PROGRAM C03_AlarmMessageControl
VAR
	bAlarmGroup0Reset 		:BOOL;
	bAlarmGroup1Reset 		:BOOL;
	bAlarmGroup2Reset 		:BOOL;
	bAlarmGroup3Reset 		:BOOL;
	bAlarmGroup4Reset 		:BOOL;
	bAlarmGroup5Reset 		:BOOL;
	bAlarmGroup6Reset 		:BOOL;
	bAlarmGroup7Reset 		:BOOL;

	fbMsg_GroupPriority0	:FB_ALARM_GroupManagment;
	fbMsg_GroupPriority1	:FB_ALARM_GroupManagment;
	fbMsg_GroupPriority2	:FB_ALARM_GroupManagment;
	fbMsg_GroupPriority3	:FB_ALARM_GroupManagment;
	fbMsg_GroupPriority4	:FB_ALARM_GroupManagment;
	fbMsg_GroupPriority5	:FB_ALARM_GroupManagment;
	fbMsg_GroupPriority6	:FB_ALARM_GroupManagment;
	fbMsg_GroupPriority7	:FB_ALARM_GroupManagment;

	fbLogTable							: FB_ALARM_LogTable;
	//fbOutputDB						: FB_ALARM_OutputDB;

	aAlarmPulse						: ARRAY[0..255] OF TP;
	aTorqueStartDelayTimer			: ARRAY[1..cMAX_PROFINET_DRIVES] OF TON;

	nAlarmIndex						: INT;
	aMsgGroupStartIndex				: ARRAY[0..10] OF INT;

	bGeneralSystemAlarmActive		: BOOL;		(*Message type 0*)
	bEUCASubsytemAlarmActive		: BOOL;		(*Message type 1*)
	bTPDSubsytemAlarmActive			: BOOL;		(*Message type 2*)
	bExternalAlarmActive			: BOOL;		(*Message type 3*)

	bSpare04AlarmActive				: BOOL;		(*Message type 4*)
	bSpare05AlarmActive				: BOOL;		(*Message type 5*)
	bSpare06AlarmActive				: BOOL;		(*Message type 6*)
	bSpare07AlarmActive				: BOOL;		(*Message type 7*)

	bGeneralSystemWarningActive		: BOOL;		(*Message type 8*)
	bEUCASubsytemWarningActive		: BOOL;		(*Message type 9*)
	bTPDSubsytemWarningActive		: BOOL;		(*Message type 10*)
	bExternalWarningActive			: BOOL;		(*Message type 11*)

	bSpare12WarningActive			: BOOL;		(*Message type 12*)
	bSpare13WarningActive			: BOOL;		(*Message type 13*)
	bSpare14WarningActive			: BOOL;		(*Message type 14*)
	bSpare15WarningActive			: BOOL;		(*Message type 15*)

END_VAR
VAR // added by the converter: edge detectors and wires of the graphical bodies
    _w1, _w2, _w3, _w4, _w5, _w6, _w7, _w8 : BOOL;
END_VAR

(****************************************************************************************)
(*
bAlarmTrigger - set true to activate message
nCategoryNo - message category number (for future purpose)
nMessageTypeNo - message type number determine active message type flag
sTextMessage - message description shown in HMI
tAlarmTimout - message became active after time delay
bAlarmDefinitionEnable - enable message block executing
bInhibitReset - set acknowledge to reset/confirm active message 
*)
(****************************************************************************************)

MsgReset();
nAlarmIndex := 0;

(****************************************************************************************)

aMsgGroupStartIndex[0] := nAlarmIndex;
Msg_000_033_General();

aMsgGroupStartIndex[1] := nAlarmIndex;
Msg_034_074_Cameras();

aMsgGroupStartIndex[2] := nAlarmIndex;
Msg_075_126_Process();

aMsgGroupStartIndex[3] := nAlarmIndex;
Msg_127_150_Sensors();

aMsgGroupStartIndex[4] := nAlarmIndex;
Msg_151_179_Doors();

aMsgGroupStartIndex[5] := nAlarmIndex;
Msg_180_200_Motors();

aMsgGroupStartIndex[6] := nAlarmIndex;
Msg_201_208_Interface();

aMsgGroupStartIndex[7] := nAlarmIndex;
Msg_209_237_Labellers();

aMsgGroupStartIndex[8] := nAlarmIndex;
Msg_238_243_Spare();

aMsgGroupStartIndex[9] := nAlarmIndex;
Msg_244_253_DB();

aMsgGroupStartIndex[10] := nAlarmIndex;
Msg_254_255_Reserved();

(****************************************************************************************)

fbMsg_GroupPriority0	(

	stAlarms 				:= gMessage.aAlarms[0],
	stAlarmsSettings		:= gMessage.aAlarmsSettings[0]

					);
(****************************************************************************************)

fbMsg_GroupPriority1	(

	stAlarms 				:= gMessage.aAlarms[1],
	stAlarmsSettings		:= gMessage.aAlarmsSettings[1],

					);
(****************************************************************************************)

fbMsg_GroupPriority2	(

	stAlarms 				:= gMessage.aAlarms[2],
	stAlarmsSettings		:= gMessage.aAlarmsSettings[2]

					);
(****************************************************************************************)

fbMsg_GroupPriority3	(

	stAlarms 				:= gMessage.aAlarms[3],
	stAlarmsSettings		:= gMessage.aAlarmsSettings[3],

					);
(****************************************************************************************)

fbMsg_GroupPriority4		(

	stAlarms 				:= gMessage.aAlarms[4],
	stAlarmsSettings		:= gMessage.aAlarmsSettings[4]

					);
(****************************************************************************************)

fbMsg_GroupPriority5	(

	stAlarms 				:= gMessage.aAlarms[5],
	stAlarmsSettings		:= gMessage.aAlarmsSettings[5]

					);
(****************************************************************************************)

fbMsg_GroupPriority6	(

	stAlarms 				:= gMessage.aAlarms[6],
	stAlarmsSettings		:= gMessage.aAlarmsSettings[6]

					);
(****************************************************************************************)

fbMsg_GroupPriority7	(

	stAlarms 				:= gMessage.aAlarms[7],
	stAlarmsSettings		:= gMessage.aAlarmsSettings[7]

					);
(**************************************************************************************************)
(**************************** **********Alarms Logger***********************************************)
(**************************************************************************************************)

fbLogTable(
			bResetActive		:= gDevice.stMetsStatus.bShortReset,
			stAlarmTable		:= gMessage.stAlarmTable,
			aAlarms 			:= gMessage.aAlarms,
			aAlarmsSettings		:= gMessage.aAlarmsSettings,
			stCTDateTime		:= gDevice.stMetsStatus.stCTDateTime
		);
		
(*fbOutputDB(
	bSystemTimeValid		:= gDevice.stMetsStatus.bSystemTimeValid,
	stCTDateTime			:= gDevice.stMetsStatus.stCTDateTime,
	nAppOnlineChangeCnt 	:= gDevice.stPLCAppSys.OnlineChangeCnt,
	stAlarmTable			:= gMessage.stAlarmTable,
	stMachineConfig			:= gDevice.stMachineConfig
	);
*)
(**************************************************************************************************)
(**************************** **********Fault Monitor***********************************************)
(**************************************************************************************************)

IF 	gMessage.aAlarms[0].nMessageType.0	OR
	gMessage.aAlarms[1].nMessageType.0	OR
	gMessage.aAlarms[2].nMessageType.0	OR
	gMessage.aAlarms[3].nMessageType.0	OR
	gMessage.aAlarms[4].nMessageType.0	OR
	gMessage.aAlarms[5].nMessageType.0	OR
	gMessage.aAlarms[6].nMessageType.0	OR
	gMessage.aAlarms[7].nMessageType.0	THEN

		gMessage.stAlarmStatus.bGeneralSystemAlarmActive	:=	TRUE;
ELSE
		gMessage.stAlarmStatus.bGeneralSystemAlarmActive	:= 	FALSE;
END_IF

IF 	gMessage.aAlarms[0].nMessageType.1	OR
	gMessage.aAlarms[1].nMessageType.1	OR
	gMessage.aAlarms[2].nMessageType.1	OR
	gMessage.aAlarms[3].nMessageType.1	OR
	gMessage.aAlarms[4].nMessageType.1	OR
	gMessage.aAlarms[5].nMessageType.1	OR
	gMessage.aAlarms[6].nMessageType.1	OR
	gMessage.aAlarms[7].nMessageType.1	THEN

		gMessage.stAlarmStatus.bEUCASubsytemAlarmActive	:=	TRUE;
ELSE
		gMessage.stAlarmStatus.bEUCASubsytemAlarmActive	:= 	FALSE;
END_IF

IF 	gMessage.aAlarms[0].nMessageType.2	OR
	gMessage.aAlarms[1].nMessageType.2	OR
	gMessage.aAlarms[2].nMessageType.2	OR
	gMessage.aAlarms[3].nMessageType.2	OR
	gMessage.aAlarms[4].nMessageType.2	OR
	gMessage.aAlarms[5].nMessageType.2	OR
	gMessage.aAlarms[6].nMessageType.2	OR
	gMessage.aAlarms[7].nMessageType.2	THEN

		gMessage.stAlarmStatus.bTPDSubsytemAlarmActive	:=	TRUE;
ELSE
		gMessage.stAlarmStatus.bTPDSubsytemAlarmActive	:= 	FALSE;
END_IF

IF 	gMessage.aAlarms[0].nMessageType.3	OR
	gMessage.aAlarms[1].nMessageType.3	OR
	gMessage.aAlarms[2].nMessageType.3	OR
	gMessage.aAlarms[3].nMessageType.3	OR
	gMessage.aAlarms[4].nMessageType.3	OR
	gMessage.aAlarms[5].nMessageType.3	OR
	gMessage.aAlarms[6].nMessageType.3	OR
	gMessage.aAlarms[7].nMessageType.3	THEN

		gMessage.stAlarmStatus.bExternalAlarmActive	:=	TRUE;
ELSE
		gMessage.stAlarmStatus.bExternalAlarmActive	:= 	FALSE;
END_IF

IF 	gMessage.aAlarms[0].nMessageType.4	OR
	gMessage.aAlarms[1].nMessageType.4	OR
	gMessage.aAlarms[2].nMessageType.4	OR
	gMessage.aAlarms[3].nMessageType.4	OR
	gMessage.aAlarms[4].nMessageType.4	OR
	gMessage.aAlarms[5].nMessageType.4	OR
	gMessage.aAlarms[6].nMessageType.4	OR
	gMessage.aAlarms[7].nMessageType.4	THEN

		gMessage.stAlarmStatus.bSpare04AlarmActive	:=	TRUE;
ELSE
		gMessage.stAlarmStatus.bSpare04AlarmActive	:= 	FALSE;
END_IF

IF 	gMessage.aAlarms[0].nMessageType.5	OR
	gMessage.aAlarms[1].nMessageType.5	OR
	gMessage.aAlarms[2].nMessageType.5	OR
	gMessage.aAlarms[3].nMessageType.5	OR
	gMessage.aAlarms[4].nMessageType.5	OR
	gMessage.aAlarms[5].nMessageType.5	OR
	gMessage.aAlarms[6].nMessageType.5	OR
	gMessage.aAlarms[7].nMessageType.5	THEN

		gMessage.stAlarmStatus.bSpare05AlarmActive	:=	TRUE;
ELSE
		gMessage.stAlarmStatus.bSpare05AlarmActive	:= 	FALSE;
END_IF

IF 	gMessage.aAlarms[0].nMessageType.6	OR
	gMessage.aAlarms[1].nMessageType.6	OR
	gMessage.aAlarms[2].nMessageType.6	OR
	gMessage.aAlarms[3].nMessageType.6	OR
	gMessage.aAlarms[4].nMessageType.6	OR
	gMessage.aAlarms[5].nMessageType.6	OR
	gMessage.aAlarms[6].nMessageType.6	OR
	gMessage.aAlarms[7].nMessageType.6	THEN

		gMessage.stAlarmStatus.bSpare06AlarmActive	:=	TRUE;
ELSE
		gMessage.stAlarmStatus.bSpare06AlarmActive	:= 	FALSE;
END_IF

IF 	gMessage.aAlarms[0].nMessageType.7	OR
	gMessage.aAlarms[1].nMessageType.7	OR
	gMessage.aAlarms[2].nMessageType.7	OR
	gMessage.aAlarms[3].nMessageType.7	OR
	gMessage.aAlarms[4].nMessageType.7	OR
	gMessage.aAlarms[5].nMessageType.7	OR
	gMessage.aAlarms[6].nMessageType.7	OR
	gMessage.aAlarms[7].nMessageType.7	THEN

		gMessage.stAlarmStatus.bSpare07AlarmActive	:=	TRUE;
ELSE
		gMessage.stAlarmStatus.bSpare07AlarmActive	:= 	FALSE;
END_IF


IF 	gMessage.aAlarms[0].nMessageType.8	OR
	gMessage.aAlarms[1].nMessageType.8	OR
	gMessage.aAlarms[2].nMessageType.8	OR
	gMessage.aAlarms[3].nMessageType.8	OR
	gMessage.aAlarms[4].nMessageType.8	OR
	gMessage.aAlarms[5].nMessageType.8	OR
	gMessage.aAlarms[6].nMessageType.8	OR
	gMessage.aAlarms[7].nMessageType.8	THEN

		gMessage.stAlarmStatus.bGeneralSystemWarningActive	:=	TRUE;
ELSE
		gMessage.stAlarmStatus.bGeneralSystemWarningActive	:= 	FALSE;
END_IF

IF 	gMessage.aAlarms[0].nMessageType.9	OR
	gMessage.aAlarms[1].nMessageType.9	OR
	gMessage.aAlarms[2].nMessageType.9	OR
	gMessage.aAlarms[3].nMessageType.9	OR
	gMessage.aAlarms[4].nMessageType.9	OR
	gMessage.aAlarms[5].nMessageType.9	OR
	gMessage.aAlarms[6].nMessageType.9	OR
	gMessage.aAlarms[7].nMessageType.9	THEN

		gMessage.stAlarmStatus.bEUCASubsytemWarningActive	:=	TRUE;
ELSE
		gMessage.stAlarmStatus.bEUCASubsytemWarningActive	:= 	FALSE;
END_IF

IF 	gMessage.aAlarms[0].nMessageType.10	OR
	gMessage.aAlarms[1].nMessageType.10	OR
	gMessage.aAlarms[2].nMessageType.10	OR
	gMessage.aAlarms[3].nMessageType.10	OR
	gMessage.aAlarms[4].nMessageType.10	OR
	gMessage.aAlarms[5].nMessageType.10	OR
	gMessage.aAlarms[6].nMessageType.10	OR
	gMessage.aAlarms[7].nMessageType.10	THEN

		gMessage.stAlarmStatus.bTPDSubsytemWarningActive	:=	TRUE;
ELSE
		gMessage.stAlarmStatus.bTPDSubsytemWarningActive	:= 	FALSE;
END_IF

IF 	gMessage.aAlarms[0].nMessageType.11	OR
	gMessage.aAlarms[1].nMessageType.11	OR
	gMessage.aAlarms[2].nMessageType.11	OR
	gMessage.aAlarms[3].nMessageType.11	OR
	gMessage.aAlarms[4].nMessageType.11	OR
	gMessage.aAlarms[5].nMessageType.11	OR
	gMessage.aAlarms[6].nMessageType.11	OR
	gMessage.aAlarms[7].nMessageType.11	THEN

		gMessage.stAlarmStatus.bExternalWarningActive	:=	TRUE;
ELSE
		gMessage.stAlarmStatus.bExternalWarningActive	:= 	FALSE;
END_IF

IF 	gMessage.aAlarms[0].nMessageType.12	OR
	gMessage.aAlarms[1].nMessageType.12	OR
	gMessage.aAlarms[2].nMessageType.12	OR
	gMessage.aAlarms[3].nMessageType.12	OR
	gMessage.aAlarms[4].nMessageType.12	OR
	gMessage.aAlarms[5].nMessageType.12	OR
	gMessage.aAlarms[6].nMessageType.12	OR
	gMessage.aAlarms[7].nMessageType.12	THEN

		gMessage.stAlarmStatus.bSpare12WarningActive	:=	TRUE;
ELSE
		gMessage.stAlarmStatus.bSpare12WarningActive	:= 	FALSE;
END_IF

IF 	gMessage.aAlarms[0].nMessageType.13	OR
	gMessage.aAlarms[1].nMessageType.13	OR
	gMessage.aAlarms[2].nMessageType.13	OR
	gMessage.aAlarms[3].nMessageType.13	OR
	gMessage.aAlarms[4].nMessageType.13	OR
	gMessage.aAlarms[5].nMessageType.13	OR
	gMessage.aAlarms[6].nMessageType.13	OR
	gMessage.aAlarms[7].nMessageType.13	THEN

		gMessage.stAlarmStatus.bSpare13WarningActive	:=	TRUE;
ELSE
		gMessage.stAlarmStatus.bSpare13WarningActive	:= 	FALSE;
END_IF

IF 	gMessage.aAlarms[0].nMessageType.14	OR
	gMessage.aAlarms[1].nMessageType.14	OR
	gMessage.aAlarms[2].nMessageType.14	OR
	gMessage.aAlarms[3].nMessageType.14	OR
	gMessage.aAlarms[4].nMessageType.14	OR
	gMessage.aAlarms[5].nMessageType.14	OR
	gMessage.aAlarms[6].nMessageType.14	OR
	gMessage.aAlarms[7].nMessageType.14	THEN

		gMessage.stAlarmStatus.bSpare14WarningActive	:=	TRUE;
ELSE
		gMessage.stAlarmStatus.bSpare14WarningActive	:= 	FALSE;
END_IF

IF 	gMessage.aAlarms[0].nMessageType.15	OR
	gMessage.aAlarms[1].nMessageType.15	OR
	gMessage.aAlarms[2].nMessageType.15	OR
	gMessage.aAlarms[3].nMessageType.15	OR
	gMessage.aAlarms[4].nMessageType.15	OR
	gMessage.aAlarms[5].nMessageType.15	OR
	gMessage.aAlarms[6].nMessageType.15	OR
	gMessage.aAlarms[7].nMessageType.15	THEN

		gMessage.stAlarmStatus.bSpare15WarningActive	:=	TRUE;
ELSE
		gMessage.stAlarmStatus.bSpare15WarningActive	:= 	FALSE;
END_IF

(**************************************************************************************************)
(**********************************Group Fault Monitor**********************************************)
(**************************************************************************************************)

(*Message type from 0 to 3 are set up as alarms - if modyfie it is neccesary change alarm definition F_ALARM_SetDefinition for AutoReset flag*)

IF 	gMessage.stAlarmStatus.bGeneralSystemAlarmActive 		OR
	gMessage.stAlarmStatus.bEUCASubsytemAlarmActive 		OR
	gMessage.stAlarmStatus.bTPDSubsytemAlarmActive			OR
	gMessage.stAlarmStatus.bExternalAlarmActive				OR
	gMessage.stAlarmStatus.bSpare04AlarmActive 				OR
	gMessage.stAlarmStatus.bSpare05AlarmActive 				OR
	gMessage.stAlarmStatus.bSpare06AlarmActive				OR
	gMessage.stAlarmStatus.bSpare07AlarmActive				THEN

		gMessage.stAlarmStatus.bNoActiveAlarms	:=	FALSE;
ELSE
		gMessage.stAlarmStatus.bNoActiveAlarms	:=	TRUE;
END_IF

(*Message type from 4 to 7 are set up as warnings - if modyfie it is neccesary change alarm definition F_ALARM_SetDefinition for AutoReset flag*)

IF 	gMessage.stAlarmStatus.bGeneralSystemWarningActive 		OR
	gMessage.stAlarmStatus.bEUCASubsytemWarningActive 	OR
	gMessage.stAlarmStatus.bTPDSubsytemWarningActive		OR
	gMessage.stAlarmStatus.bExternalWarningActive			OR
	gMessage.stAlarmStatus.bSpare12WarningActive 			OR
	gMessage.stAlarmStatus.bSpare13WarningActive 			OR
	gMessage.stAlarmStatus.bSpare14WarningActive			OR
	gMessage.stAlarmStatus.bSpare15WarningActive			THEN

		gMessage.stAlarmStatus.bNoActiveWarrnings	:=	FALSE;
ELSE
		gMessage.stAlarmStatus.bNoActiveWarrnings	:=	TRUE;
END_IF

ACTION Msg_000_033_General:
// note: this text did not pass the execution check against the stored diagram
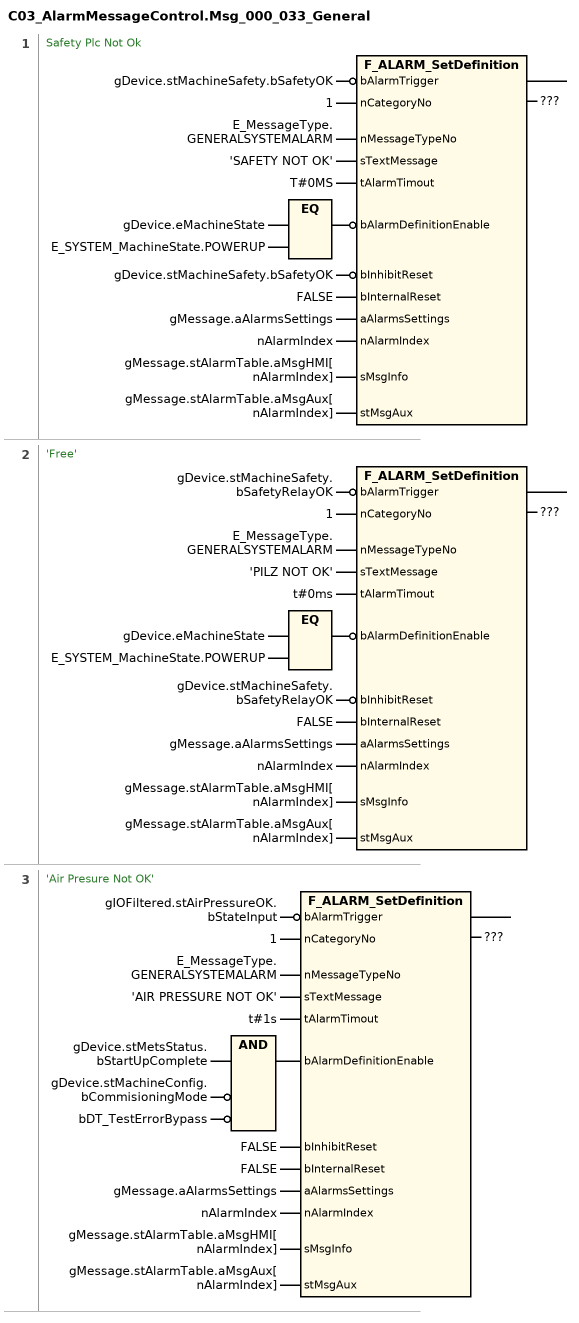
// NETWORK 1
//  Safety Plc Not Ok
F_ALARM_SetDefinition(bAlarmTrigger := NOT gDevice.stMachineSafety.bSafetyOK, nCategoryNo := 1, nMessageTypeNo := E_MessageType.GENERALSYSTEMALARM, sTextMessage := 'SAFETY NOT OK', tAlarmTimout := T#0MS, bAlarmDefinitionEnable := NOT (gDevice.eMachineState = E_SYSTEM_MachineState.POWERUP), bInhibitReset := NOT gDevice.stMachineSafety.bSafetyOK, bInternalReset := FALSE, aAlarmsSettings := gMessage.aAlarmsSettings, nAlarmIndex := nAlarmIndex, sMsgInfo := gMessage.stAlarmTable.aMsgHMI[nAlarmIndex], stMsgAux := gMessage.stAlarmTable.aMsgAux[nAlarmIndex]);

// NETWORK 2
// 'Free'
F_ALARM_SetDefinition(bAlarmTrigger := NOT gDevice.stMachineSafety.bSafetyRelayOK, nCategoryNo := 1, nMessageTypeNo := E_MessageType.GENERALSYSTEMALARM, sTextMessage := 'PILZ NOT OK', tAlarmTimout := t#0ms, bAlarmDefinitionEnable := NOT (gDevice.eMachineState = E_SYSTEM_MachineState.POWERUP), bInhibitReset := NOT gDevice.stMachineSafety.bSafetyRelayOK, bInternalReset := FALSE, aAlarmsSettings := gMessage.aAlarmsSettings, nAlarmIndex := nAlarmIndex, sMsgInfo := gMessage.stAlarmTable.aMsgHMI[nAlarmIndex], stMsgAux := gMessage.stAlarmTable.aMsgAux[nAlarmIndex]);

// NETWORK 3
// 'Air Presure Not OK'
F_ALARM_SetDefinition(bAlarmTrigger := NOT gIOFiltered.stAirPressureOK.bStateInput, nCategoryNo := 1, nMessageTypeNo := E_MessageType.GENERALSYSTEMALARM, sTextMessage := 'AIR PRESSURE NOT OK', tAlarmTimout := t#1s, bAlarmDefinitionEnable := gDevice.stMetsStatus.bStartUpComplete AND NOT gDevice.stMachineConfig.bCommisioningMode AND NOT bDT_TestErrorBypass, bInhibitReset := FALSE, bInternalReset := FALSE, aAlarmsSettings := gMessage.aAlarmsSettings, nAlarmIndex := nAlarmIndex, sMsgInfo := gMessage.stAlarmTable.aMsgHMI[nAlarmIndex], stMsgAux := gMessage.stAlarmTable.aMsgAux[nAlarmIndex]);

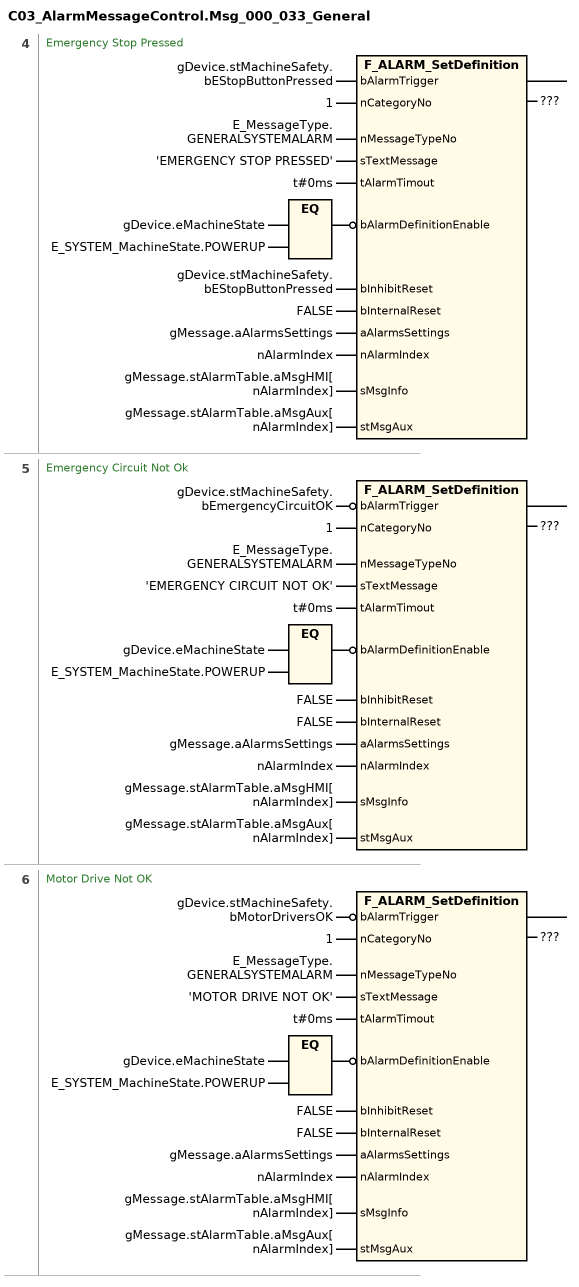
// NETWORK 4
// 					Emergency Stop Pressed
//
//
F_ALARM_SetDefinition(bAlarmTrigger := gDevice.stMachineSafety.bEStopButtonPressed, nCategoryNo := 1, nMessageTypeNo := E_MessageType.GENERALSYSTEMALARM, sTextMessage := 'EMERGENCY STOP PRESSED', tAlarmTimout := t#0ms, bAlarmDefinitionEnable := NOT (gDevice.eMachineState = E_SYSTEM_MachineState.POWERUP), bInhibitReset := gDevice.stMachineSafety.bEStopButtonPressed, bInternalReset := FALSE, aAlarmsSettings := gMessage.aAlarmsSettings, nAlarmIndex := nAlarmIndex, sMsgInfo := gMessage.stAlarmTable.aMsgHMI[nAlarmIndex], stMsgAux := gMessage.stAlarmTable.aMsgAux[nAlarmIndex]);

// NETWORK 5
// 					Emergency Circuit Not Ok
//
//
F_ALARM_SetDefinition(bAlarmTrigger := NOT gDevice.stMachineSafety.bEmergencyCircuitOK, nCategoryNo := 1, nMessageTypeNo := E_MessageType.GENERALSYSTEMALARM, sTextMessage := 'EMERGENCY CIRCUIT NOT OK', tAlarmTimout := t#0ms, bAlarmDefinitionEnable := NOT (gDevice.eMachineState = E_SYSTEM_MachineState.POWERUP), bInhibitReset := FALSE, bInternalReset := FALSE, aAlarmsSettings := gMessage.aAlarmsSettings, nAlarmIndex := nAlarmIndex, sMsgInfo := gMessage.stAlarmTable.aMsgHMI[nAlarmIndex], stMsgAux := gMessage.stAlarmTable.aMsgAux[nAlarmIndex]);

// NETWORK 6
// 					Motor Drive Not OK
//
//
F_ALARM_SetDefinition(bAlarmTrigger := NOT gDevice.stMachineSafety.bMotorDriversOK, nCategoryNo := 1, nMessageTypeNo := E_MessageType.GENERALSYSTEMALARM, sTextMessage := 'MOTOR DRIVE NOT OK', tAlarmTimout := t#0ms, bAlarmDefinitionEnable := NOT (gDevice.eMachineState = E_SYSTEM_MachineState.POWERUP), bInhibitReset := FALSE, bInternalReset := FALSE, aAlarmsSettings := gMessage.aAlarmsSettings, nAlarmIndex := nAlarmIndex, sMsgInfo := gMessage.stAlarmTable.aMsgHMI[nAlarmIndex], stMsgAux := gMessage.stAlarmTable.aMsgAux[nAlarmIndex]);

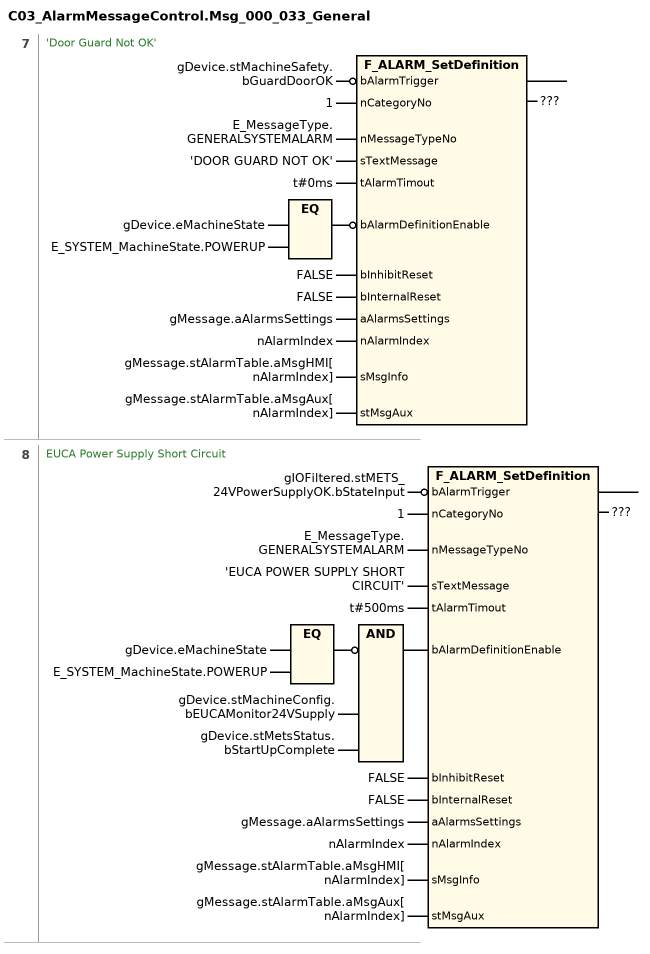
// NETWORK 7
// 					'Door Guard Not OK'
//
//
F_ALARM_SetDefinition(bAlarmTrigger := NOT gDevice.stMachineSafety.bGuardDoorOK, nCategoryNo := 1, nMessageTypeNo := E_MessageType.GENERALSYSTEMALARM, sTextMessage := 'DOOR GUARD NOT OK', tAlarmTimout := t#0ms, bAlarmDefinitionEnable := NOT (gDevice.eMachineState = E_SYSTEM_MachineState.POWERUP), bInhibitReset := FALSE, bInternalReset := FALSE, aAlarmsSettings := gMessage.aAlarmsSettings, nAlarmIndex := nAlarmIndex, sMsgInfo := gMessage.stAlarmTable.aMsgHMI[nAlarmIndex], stMsgAux := gMessage.stAlarmTable.aMsgAux[nAlarmIndex]);

// NETWORK 8
// EUCA Power Supply Short Circuit
F_ALARM_SetDefinition(bAlarmTrigger := NOT gIOFiltered.stMETS_24VPowerSupplyOK.bStateInput, nCategoryNo := 1, nMessageTypeNo := E_MessageType.GENERALSYSTEMALARM, sTextMessage := 'EUCA POWER SUPPLY SHORT CIRCUIT', tAlarmTimout := t#500ms, bAlarmDefinitionEnable := NOT (gDevice.eMachineState = E_SYSTEM_MachineState.POWERUP) AND gDevice.stMachineConfig.bEUCAMonitor24VSupply AND gDevice.stMetsStatus.bStartUpComplete, bInhibitReset := FALSE, bInternalReset := FALSE, aAlarmsSettings := gMessage.aAlarmsSettings, nAlarmIndex := nAlarmIndex, sMsgInfo := gMessage.stAlarmTable.aMsgHMI[nAlarmIndex], stMsgAux := gMessage.stAlarmTable.aMsgAux[nAlarmIndex]);

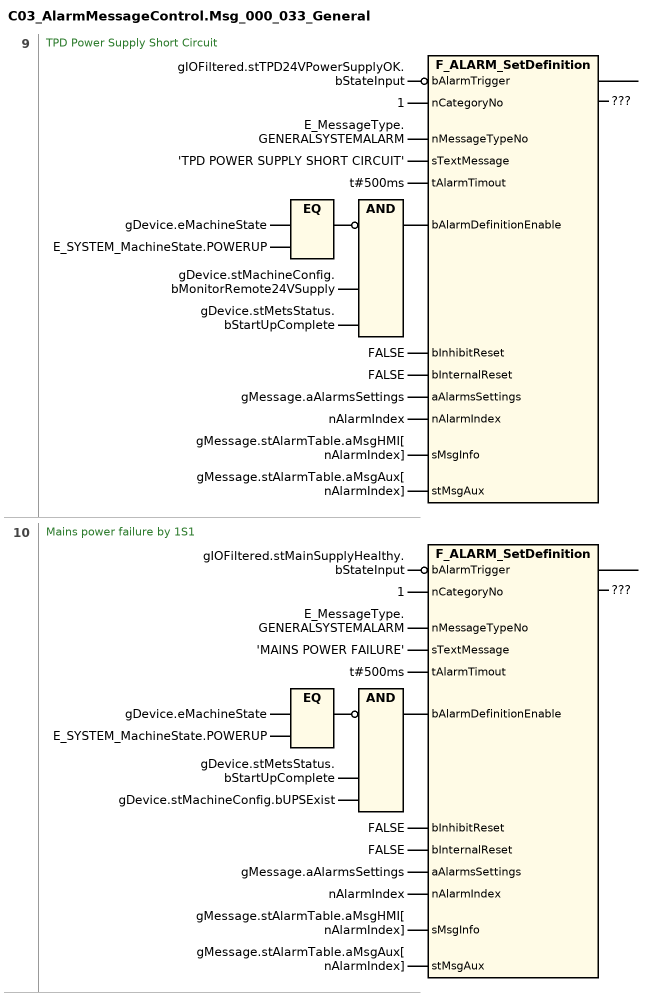
// NETWORK 9
// TPD Power Supply Short Circuit
F_ALARM_SetDefinition(bAlarmTrigger := NOT gIOFiltered.stTPD24VPowerSupplyOK.bStateInput, nCategoryNo := 1, nMessageTypeNo := E_MessageType.GENERALSYSTEMALARM, sTextMessage := 'TPD POWER SUPPLY SHORT CIRCUIT', tAlarmTimout := t#500ms, bAlarmDefinitionEnable := NOT (gDevice.eMachineState = E_SYSTEM_MachineState.POWERUP) AND gDevice.stMachineConfig.bMonitorRemote24VSupply AND gDevice.stMetsStatus.bStartUpComplete, bInhibitReset := FALSE, bInternalReset := FALSE, aAlarmsSettings := gMessage.aAlarmsSettings, nAlarmIndex := nAlarmIndex, sMsgInfo := gMessage.stAlarmTable.aMsgHMI[nAlarmIndex], stMsgAux := gMessage.stAlarmTable.aMsgAux[nAlarmIndex]);

// NETWORK 10
// Mains power failure by 1S1
F_ALARM_SetDefinition(bAlarmTrigger := NOT gIOFiltered.stMainSupplyHealthy.bStateInput, nCategoryNo := 1, nMessageTypeNo := E_MessageType.GENERALSYSTEMALARM, sTextMessage := 'MAINS POWER FAILURE', tAlarmTimout := t#500ms, bAlarmDefinitionEnable := NOT (gDevice.eMachineState = E_SYSTEM_MachineState.POWERUP) AND gDevice.stMetsStatus.bStartUpComplete AND gDevice.stMachineConfig.bUPSExist, bInhibitReset := FALSE, bInternalReset := FALSE, aAlarmsSettings := gMessage.aAlarmsSettings, nAlarmIndex := nAlarmIndex, sMsgInfo := gMessage.stAlarmTable.aMsgHMI[nAlarmIndex], stMsgAux := gMessage.stAlarmTable.aMsgAux[nAlarmIndex]);

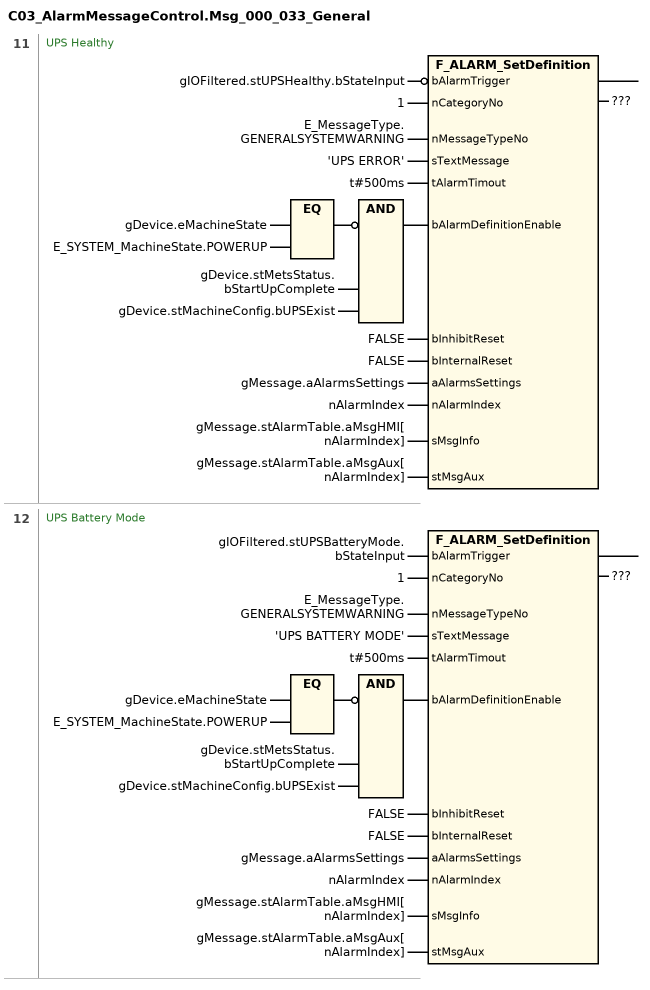
// NETWORK 11
// UPS Healthy
F_ALARM_SetDefinition(bAlarmTrigger := NOT gIOFiltered.stUPSHealthy.bStateInput, nCategoryNo := 1, nMessageTypeNo := E_MessageType.GENERALSYSTEMWARNING, sTextMessage := 'UPS ERROR', tAlarmTimout := t#500ms, bAlarmDefinitionEnable := NOT (gDevice.eMachineState = E_SYSTEM_MachineState.POWERUP) AND gDevice.stMetsStatus.bStartUpComplete AND gDevice.stMachineConfig.bUPSExist, bInhibitReset := FALSE, bInternalReset := FALSE, aAlarmsSettings := gMessage.aAlarmsSettings, nAlarmIndex := nAlarmIndex, sMsgInfo := gMessage.stAlarmTable.aMsgHMI[nAlarmIndex], stMsgAux := gMessage.stAlarmTable.aMsgAux[nAlarmIndex]);

// NETWORK 12
// UPS Battery Mode
F_ALARM_SetDefinition(bAlarmTrigger := gIOFiltered.stUPSBatteryMode.bStateInput, nCategoryNo := 1, nMessageTypeNo := E_MessageType.GENERALSYSTEMWARNING, sTextMessage := 'UPS BATTERY MODE', tAlarmTimout := t#500ms, bAlarmDefinitionEnable := NOT (gDevice.eMachineState = E_SYSTEM_MachineState.POWERUP) AND gDevice.stMetsStatus.bStartUpComplete AND gDevice.stMachineConfig.bUPSExist, bInhibitReset := FALSE, bInternalReset := FALSE, aAlarmsSettings := gMessage.aAlarmsSettings, nAlarmIndex := nAlarmIndex, sMsgInfo := gMessage.stAlarmTable.aMsgHMI[nAlarmIndex], stMsgAux := gMessage.stAlarmTable.aMsgAux[nAlarmIndex]);

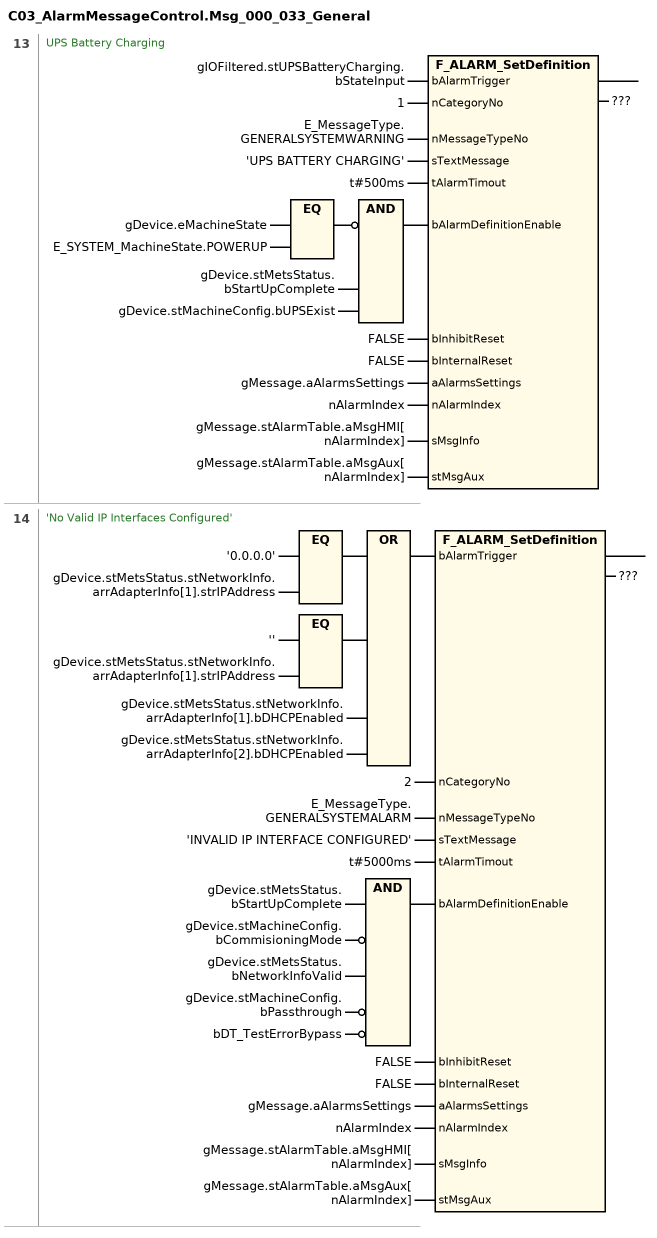
// NETWORK 13
// UPS Battery Charging
F_ALARM_SetDefinition(bAlarmTrigger := gIOFiltered.stUPSBatteryCharging.bStateInput, nCategoryNo := 1, nMessageTypeNo := E_MessageType.GENERALSYSTEMWARNING, sTextMessage := 'UPS BATTERY CHARGING', tAlarmTimout := t#500ms, bAlarmDefinitionEnable := NOT (gDevice.eMachineState = E_SYSTEM_MachineState.POWERUP) AND gDevice.stMetsStatus.bStartUpComplete AND gDevice.stMachineConfig.bUPSExist, bInhibitReset := FALSE, bInternalReset := FALSE, aAlarmsSettings := gMessage.aAlarmsSettings, nAlarmIndex := nAlarmIndex, sMsgInfo := gMessage.stAlarmTable.aMsgHMI[nAlarmIndex], stMsgAux := gMessage.stAlarmTable.aMsgAux[nAlarmIndex]);

// NETWORK 14
// 'No Valid IP Interfaces Configured'
F_ALARM_SetDefinition(bAlarmTrigger := '0.0.0.0' = gDevice.stMetsStatus.stNetworkInfo.arrAdapterInfo[1].strIPAddress OR '' = gDevice.stMetsStatus.stNetworkInfo.arrAdapterInfo[1].strIPAddress OR gDevice.stMetsStatus.stNetworkInfo.arrAdapterInfo[1].bDHCPEnabled OR gDevice.stMetsStatus.stNetworkInfo.arrAdapterInfo[2].bDHCPEnabled, nCategoryNo := 2, nMessageTypeNo := E_MessageType.GENERALSYSTEMALARM, sTextMessage := 'INVALID IP INTERFACE CONFIGURED', tAlarmTimout := t#5000ms, bAlarmDefinitionEnable := gDevice.stMetsStatus.bStartUpComplete AND NOT gDevice.stMachineConfig.bCommisioningMode AND gDevice.stMetsStatus.bNetworkInfoValid AND NOT gDevice.stMachineConfig.bPassthrough AND NOT bDT_TestErrorBypass, bInhibitReset := FALSE, bInternalReset := FALSE, aAlarmsSettings := gMessage.aAlarmsSettings, nAlarmIndex := nAlarmIndex, sMsgInfo := gMessage.stAlarmTable.aMsgHMI[nAlarmIndex], stMsgAux := gMessage.stAlarmTable.aMsgAux[nAlarmIndex]);

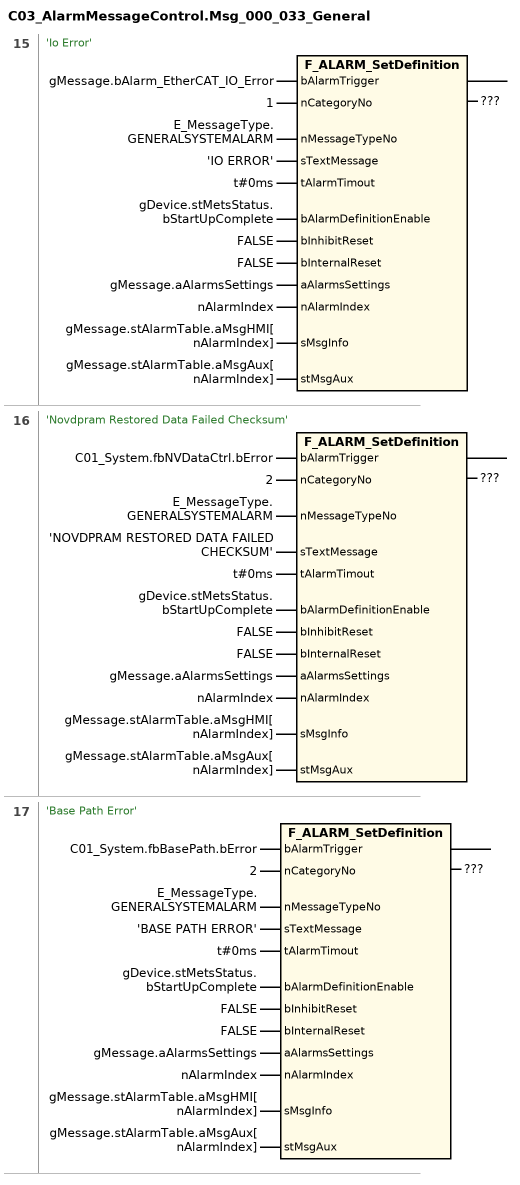
// NETWORK 15
// 'Io Error'
F_ALARM_SetDefinition(bAlarmTrigger := gMessage.bAlarm_EtherCAT_IO_Error, nCategoryNo := 1, nMessageTypeNo := E_MessageType.GENERALSYSTEMALARM, sTextMessage := 'IO ERROR', tAlarmTimout := t#0ms, bAlarmDefinitionEnable := gDevice.stMetsStatus.bStartUpComplete, bInhibitReset := FALSE, bInternalReset := FALSE, aAlarmsSettings := gMessage.aAlarmsSettings, nAlarmIndex := nAlarmIndex, sMsgInfo := gMessage.stAlarmTable.aMsgHMI[nAlarmIndex], stMsgAux := gMessage.stAlarmTable.aMsgAux[nAlarmIndex]);

// NETWORK 16
// 'Novdpram Restored Data Failed Checksum'
F_ALARM_SetDefinition(bAlarmTrigger := C01_System.fbNVDataCtrl.bError, nCategoryNo := 2, nMessageTypeNo := E_MessageType.GENERALSYSTEMALARM, sTextMessage := 'NOVDPRAM RESTORED DATA FAILED CHECKSUM', tAlarmTimout := t#0ms, bAlarmDefinitionEnable := gDevice.stMetsStatus.bStartUpComplete, bInhibitReset := FALSE, bInternalReset := FALSE, aAlarmsSettings := gMessage.aAlarmsSettings, nAlarmIndex := nAlarmIndex, sMsgInfo := gMessage.stAlarmTable.aMsgHMI[nAlarmIndex], stMsgAux := gMessage.stAlarmTable.aMsgAux[nAlarmIndex]);

// NETWORK 17
// 					'Base Path Error'
//
//
F_ALARM_SetDefinition(bAlarmTrigger := C01_System.fbBasePath.bError, nCategoryNo := 2, nMessageTypeNo := E_MessageType.GENERALSYSTEMALARM, sTextMessage := 'BASE PATH ERROR', tAlarmTimout := t#0ms, bAlarmDefinitionEnable := gDevice.stMetsStatus.bStartUpComplete, bInhibitReset := FALSE, bInternalReset := FALSE, aAlarmsSettings := gMessage.aAlarmsSettings, nAlarmIndex := nAlarmIndex, sMsgInfo := gMessage.stAlarmTable.aMsgHMI[nAlarmIndex], stMsgAux := gMessage.stAlarmTable.aMsgAux[nAlarmIndex]);

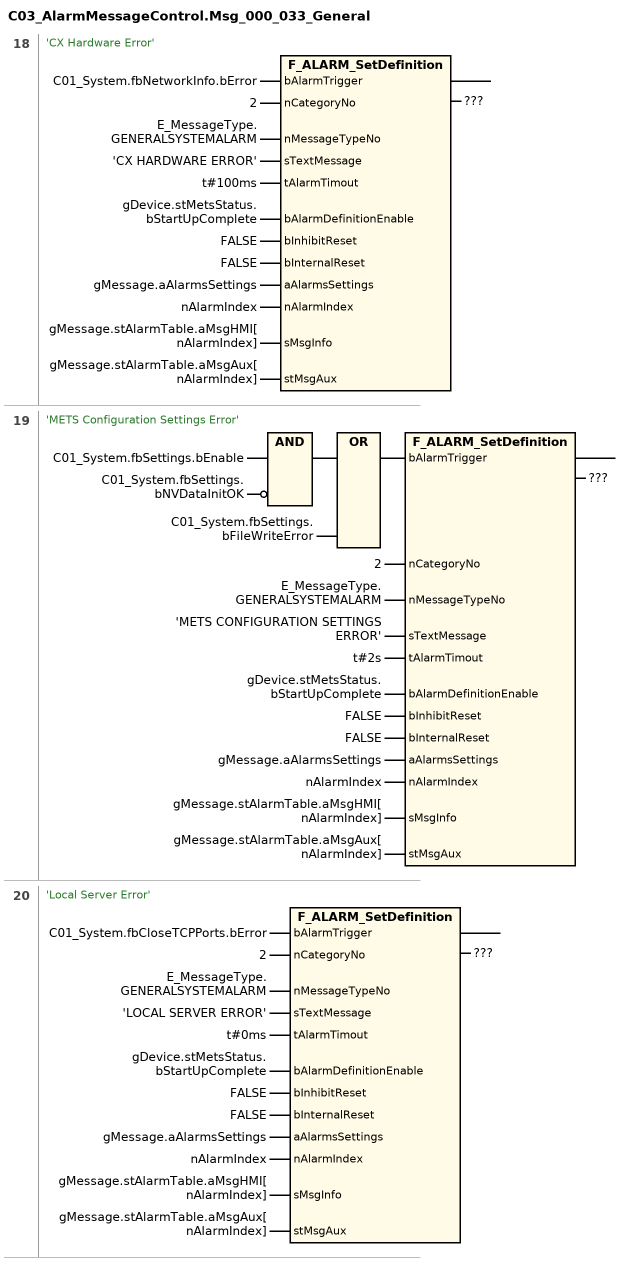
// NETWORK 18
// 					'CX Hardware Error'
//
//
F_ALARM_SetDefinition(bAlarmTrigger := C01_System.fbNetworkInfo.bError, nCategoryNo := 2, nMessageTypeNo := E_MessageType.GENERALSYSTEMALARM, sTextMessage := 'CX HARDWARE ERROR', tAlarmTimout := t#100ms, bAlarmDefinitionEnable := gDevice.stMetsStatus.bStartUpComplete, bInhibitReset := FALSE, bInternalReset := FALSE, aAlarmsSettings := gMessage.aAlarmsSettings, nAlarmIndex := nAlarmIndex, sMsgInfo := gMessage.stAlarmTable.aMsgHMI[nAlarmIndex], stMsgAux := gMessage.stAlarmTable.aMsgAux[nAlarmIndex]);

// NETWORK 19
// 'METS Configuration Settings Error'
F_ALARM_SetDefinition(bAlarmTrigger := C01_System.fbSettings.bEnable AND NOT C01_System.fbSettings.bNVDataInitOK OR C01_System.fbSettings.bFileWriteError, nCategoryNo := 2, nMessageTypeNo := E_MessageType.GENERALSYSTEMALARM, sTextMessage := 'METS CONFIGURATION SETTINGS ERROR', tAlarmTimout := t#2s, bAlarmDefinitionEnable := gDevice.stMetsStatus.bStartUpComplete, bInhibitReset := FALSE, bInternalReset := FALSE, aAlarmsSettings := gMessage.aAlarmsSettings, nAlarmIndex := nAlarmIndex, sMsgInfo := gMessage.stAlarmTable.aMsgHMI[nAlarmIndex], stMsgAux := gMessage.stAlarmTable.aMsgAux[nAlarmIndex]);

// NETWORK 20
// 					'Local Server Error'
//
//
F_ALARM_SetDefinition(bAlarmTrigger := C01_System.fbCloseTCPPorts.bError, nCategoryNo := 2, nMessageTypeNo := E_MessageType.GENERALSYSTEMALARM, sTextMessage := 'LOCAL SERVER ERROR', tAlarmTimout := t#0ms, bAlarmDefinitionEnable := gDevice.stMetsStatus.bStartUpComplete, bInhibitReset := FALSE, bInternalReset := FALSE, aAlarmsSettings := gMessage.aAlarmsSettings, nAlarmIndex := nAlarmIndex, sMsgInfo := gMessage.stAlarmTable.aMsgHMI[nAlarmIndex], stMsgAux := gMessage.stAlarmTable.aMsgAux[nAlarmIndex]);

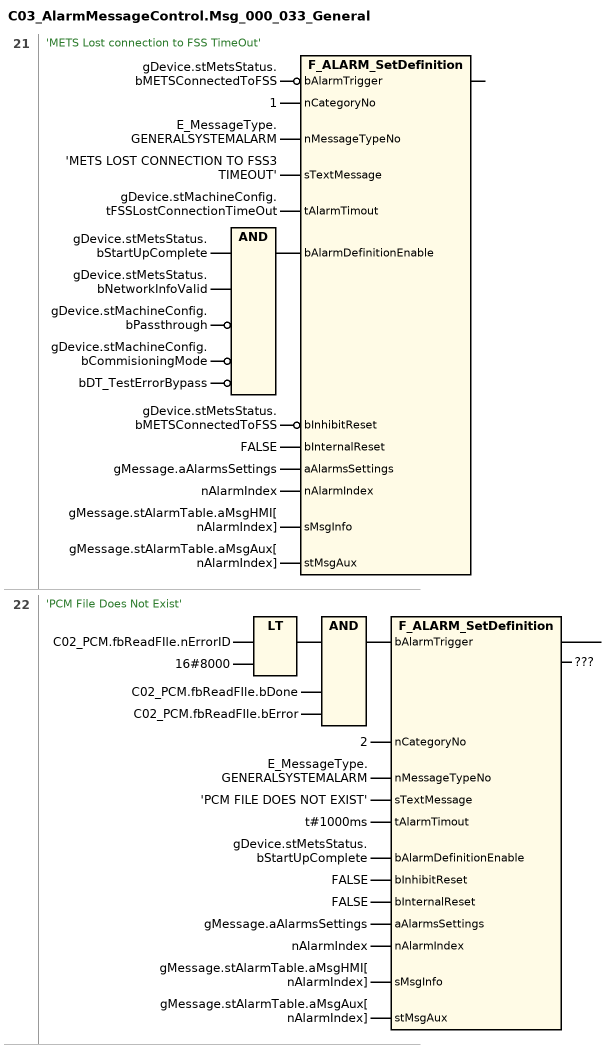
// NETWORK 21
// 'METS Lost connection to FSS TimeOut'
F_ALARM_SetDefinition(bAlarmTrigger := NOT gDevice.stMetsStatus.bMETSConnectedToFSS, nCategoryNo := 1, nMessageTypeNo := E_MessageType.GENERALSYSTEMALARM, sTextMessage := 'METS LOST CONNECTION TO FSS3 TIMEOUT', tAlarmTimout := gDevice.stMachineConfig.tFSSLostConnectionTimeOut, bAlarmDefinitionEnable := gDevice.stMetsStatus.bStartUpComplete AND gDevice.stMetsStatus.bNetworkInfoValid AND NOT gDevice.stMachineConfig.bPassthrough AND NOT gDevice.stMachineConfig.bCommisioningMode AND NOT bDT_TestErrorBypass, bInhibitReset := NOT gDevice.stMetsStatus.bMETSConnectedToFSS, bInternalReset := FALSE, aAlarmsSettings := gMessage.aAlarmsSettings, nAlarmIndex := nAlarmIndex, sMsgInfo := gMessage.stAlarmTable.aMsgHMI[nAlarmIndex], stMsgAux := gMessage.stAlarmTable.aMsgAux[nAlarmIndex]);

// NETWORK 22
// 'PCM File Does Not Exist'
F_ALARM_SetDefinition(bAlarmTrigger := C02_PCM.fbReadFIle.nErrorID < 16#8000 AND C02_PCM.fbReadFIle.bDone AND C02_PCM.fbReadFIle.bError, nCategoryNo := 2, nMessageTypeNo := E_MessageType.GENERALSYSTEMALARM, sTextMessage := 'PCM FILE DOES NOT EXIST', tAlarmTimout := t#1000ms, bAlarmDefinitionEnable := gDevice.stMetsStatus.bStartUpComplete, bInhibitReset := FALSE, bInternalReset := FALSE, aAlarmsSettings := gMessage.aAlarmsSettings, nAlarmIndex := nAlarmIndex, sMsgInfo := gMessage.stAlarmTable.aMsgHMI[nAlarmIndex], stMsgAux := gMessage.stAlarmTable.aMsgAux[nAlarmIndex]);

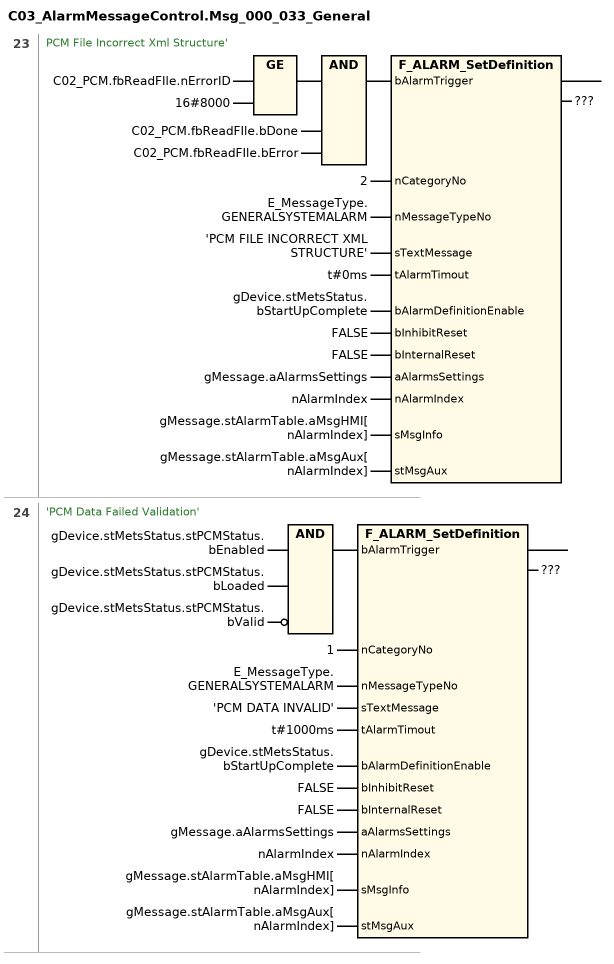
// NETWORK 23
// PCM File Incorrect Xml Structure'
F_ALARM_SetDefinition(bAlarmTrigger := C02_PCM.fbReadFIle.nErrorID >= 16#8000 AND C02_PCM.fbReadFIle.bDone AND C02_PCM.fbReadFIle.bError, nCategoryNo := 2, nMessageTypeNo := E_MessageType.GENERALSYSTEMALARM, sTextMessage := 'PCM FILE INCORRECT XML STRUCTURE', tAlarmTimout := t#0ms, bAlarmDefinitionEnable := gDevice.stMetsStatus.bStartUpComplete, bInhibitReset := FALSE, bInternalReset := FALSE, aAlarmsSettings := gMessage.aAlarmsSettings, nAlarmIndex := nAlarmIndex, sMsgInfo := gMessage.stAlarmTable.aMsgHMI[nAlarmIndex], stMsgAux := gMessage.stAlarmTable.aMsgAux[nAlarmIndex]);

// NETWORK 24
// 'PCM Data Failed Validation'
F_ALARM_SetDefinition(bAlarmTrigger := gDevice.stMetsStatus.stPCMStatus.bEnabled AND gDevice.stMetsStatus.stPCMStatus.bLoaded AND NOT gDevice.stMetsStatus.stPCMStatus.bValid, nCategoryNo := 1, nMessageTypeNo := E_MessageType.GENERALSYSTEMALARM, sTextMessage := 'PCM DATA INVALID', tAlarmTimout := t#1000ms, bAlarmDefinitionEnable := gDevice.stMetsStatus.bStartUpComplete, bInhibitReset := FALSE, bInternalReset := FALSE, aAlarmsSettings := gMessage.aAlarmsSettings, nAlarmIndex := nAlarmIndex, sMsgInfo := gMessage.stAlarmTable.aMsgHMI[nAlarmIndex], stMsgAux := gMessage.stAlarmTable.aMsgAux[nAlarmIndex]);

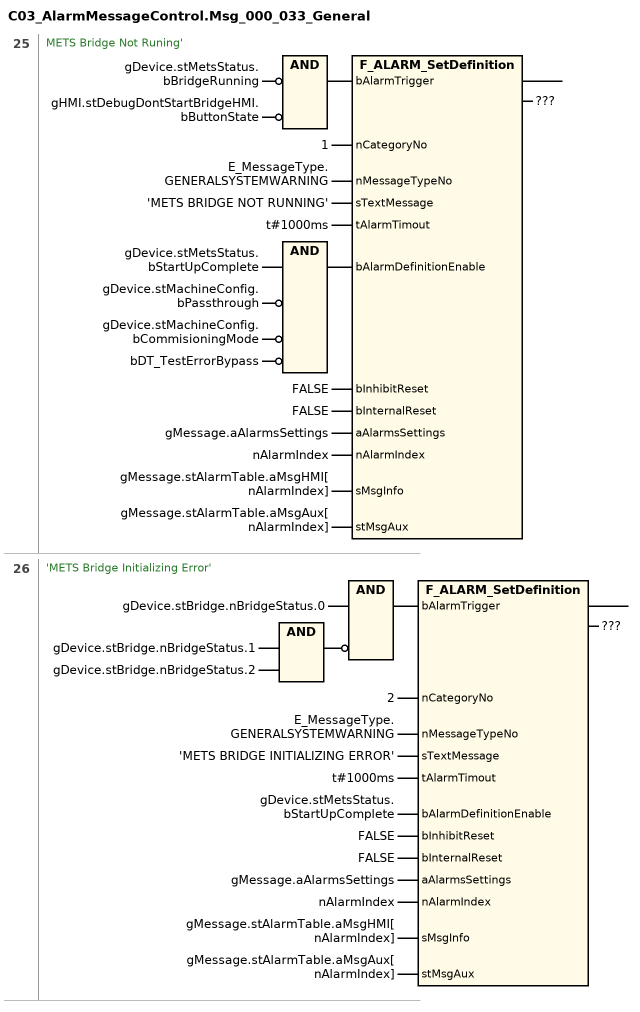
// NETWORK 25
// 					METS Bridge Not Runing'
//
//
F_ALARM_SetDefinition(bAlarmTrigger := NOT gDevice.stMetsStatus.bBridgeRunning AND NOT gHMI.stDebugDontStartBridgeHMI.bButtonState, nCategoryNo := 1, nMessageTypeNo := E_MessageType.GENERALSYSTEMWARNING, sTextMessage := 'METS BRIDGE NOT RUNNING', tAlarmTimout := t#1000ms, bAlarmDefinitionEnable := gDevice.stMetsStatus.bStartUpComplete AND NOT gDevice.stMachineConfig.bPassthrough AND NOT gDevice.stMachineConfig.bCommisioningMode AND NOT bDT_TestErrorBypass, bInhibitReset := FALSE, bInternalReset := FALSE, aAlarmsSettings := gMessage.aAlarmsSettings, nAlarmIndex := nAlarmIndex, sMsgInfo := gMessage.stAlarmTable.aMsgHMI[nAlarmIndex], stMsgAux := gMessage.stAlarmTable.aMsgAux[nAlarmIndex]);

// NETWORK 26
// 'METS Bridge Initializing Error'
F_ALARM_SetDefinition(bAlarmTrigger := gDevice.stBridge.nBridgeStatus.0 AND NOT (gDevice.stBridge.nBridgeStatus.1 AND gDevice.stBridge.nBridgeStatus.2), nCategoryNo := 2, nMessageTypeNo := E_MessageType.GENERALSYSTEMWARNING, sTextMessage := 'METS BRIDGE INITIALIZING ERROR', tAlarmTimout := t#1000ms, bAlarmDefinitionEnable := gDevice.stMetsStatus.bStartUpComplete, bInhibitReset := FALSE, bInternalReset := FALSE, aAlarmsSettings := gMessage.aAlarmsSettings, nAlarmIndex := nAlarmIndex, sMsgInfo := gMessage.stAlarmTable.aMsgHMI[nAlarmIndex], stMsgAux := gMessage.stAlarmTable.aMsgAux[nAlarmIndex]);

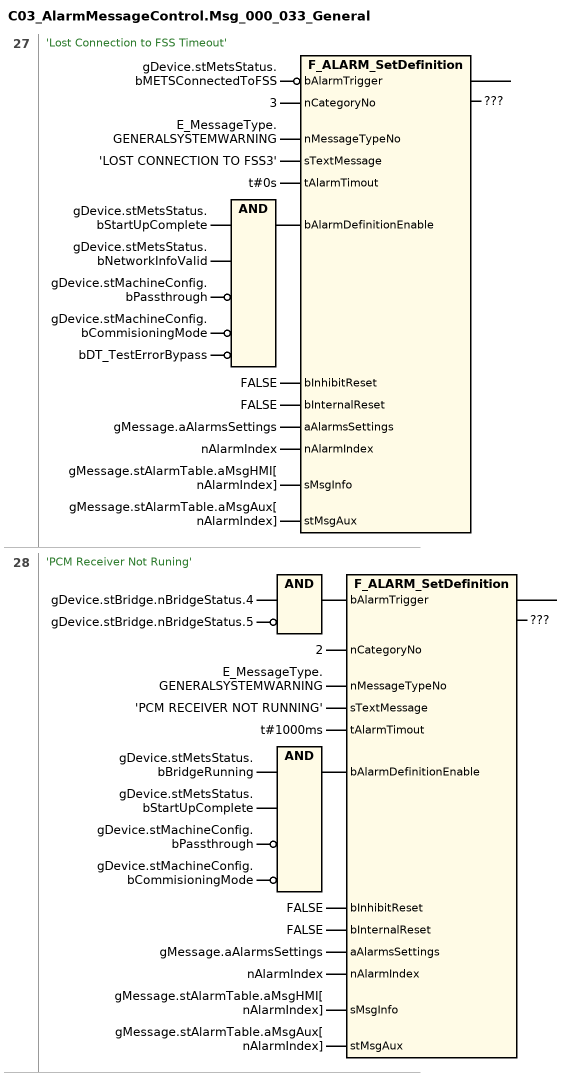
// NETWORK 27
// 'Lost Connection to FSS Timeout'
F_ALARM_SetDefinition(bAlarmTrigger := NOT gDevice.stMetsStatus.bMETSConnectedToFSS, nCategoryNo := 3, nMessageTypeNo := E_MessageType.GENERALSYSTEMWARNING, sTextMessage := 'LOST CONNECTION TO FSS3', tAlarmTimout := t#0s, bAlarmDefinitionEnable := gDevice.stMetsStatus.bStartUpComplete AND gDevice.stMetsStatus.bNetworkInfoValid AND NOT gDevice.stMachineConfig.bPassthrough AND NOT gDevice.stMachineConfig.bCommisioningMode AND NOT bDT_TestErrorBypass, bInhibitReset := FALSE, bInternalReset := FALSE, aAlarmsSettings := gMessage.aAlarmsSettings, nAlarmIndex := nAlarmIndex, sMsgInfo := gMessage.stAlarmTable.aMsgHMI[nAlarmIndex], stMsgAux := gMessage.stAlarmTable.aMsgAux[nAlarmIndex]);

// NETWORK 28
// 					'PCM Receiver Not Runing'
//
//
F_ALARM_SetDefinition(bAlarmTrigger := gDevice.stBridge.nBridgeStatus.4 AND NOT gDevice.stBridge.nBridgeStatus.5, nCategoryNo := 2, nMessageTypeNo := E_MessageType.GENERALSYSTEMWARNING, sTextMessage := 'PCM RECEIVER NOT RUNNING', tAlarmTimout := t#1000ms, bAlarmDefinitionEnable := gDevice.stMetsStatus.bBridgeRunning AND gDevice.stMetsStatus.bStartUpComplete AND NOT gDevice.stMachineConfig.bPassthrough AND NOT gDevice.stMachineConfig.bCommisioningMode, bInhibitReset := FALSE, bInternalReset := FALSE, aAlarmsSettings := gMessage.aAlarmsSettings, nAlarmIndex := nAlarmIndex, sMsgInfo := gMessage.stAlarmTable.aMsgHMI[nAlarmIndex], stMsgAux := gMessage.stAlarmTable.aMsgAux[nAlarmIndex]);

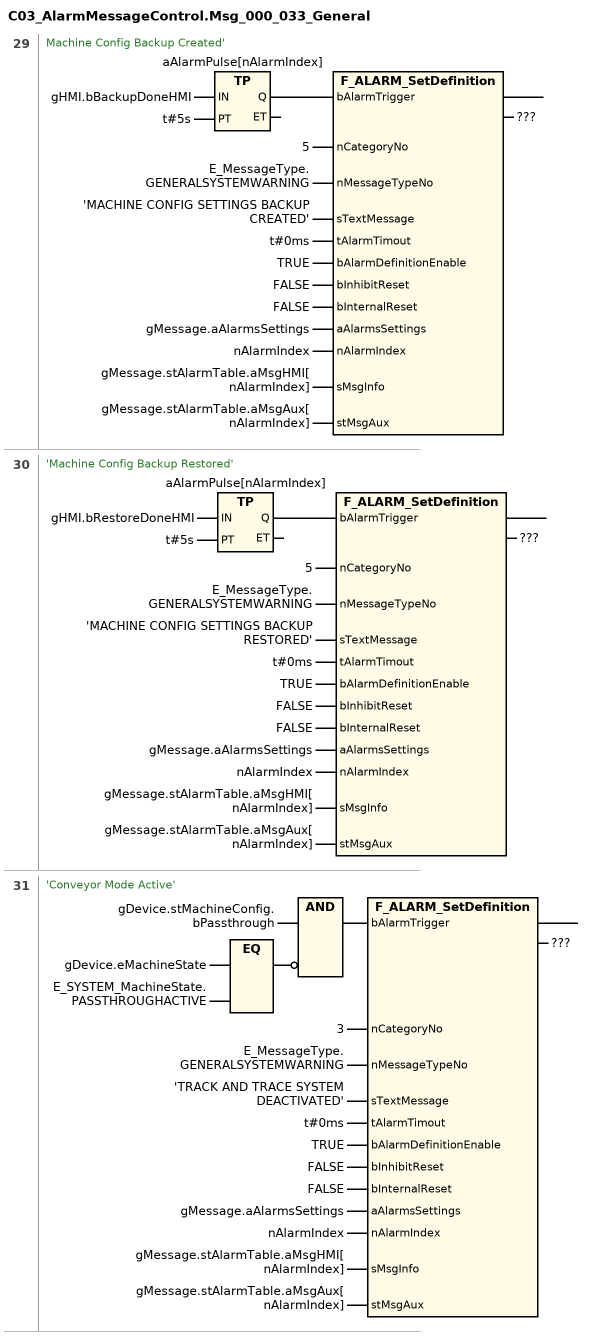
// NETWORK 29
// Machine Config Backup Created'
aAlarmPulse[nAlarmIndex](IN := gHMI.bBackupDoneHMI, PT := t#5s); // TP
F_ALARM_SetDefinition(bAlarmTrigger := aAlarmPulse[nAlarmIndex].Q, nCategoryNo := 5, nMessageTypeNo := E_MessageType.GENERALSYSTEMWARNING, sTextMessage := 'MACHINE CONFIG SETTINGS BACKUP CREATED', tAlarmTimout := t#0ms, bAlarmDefinitionEnable := TRUE, bInhibitReset := FALSE, bInternalReset := FALSE, aAlarmsSettings := gMessage.aAlarmsSettings, nAlarmIndex := nAlarmIndex, sMsgInfo := gMessage.stAlarmTable.aMsgHMI[nAlarmIndex], stMsgAux := gMessage.stAlarmTable.aMsgAux[nAlarmIndex]);

// NETWORK 30
// 'Machine Config Backup Restored'
aAlarmPulse[nAlarmIndex](IN := gHMI.bRestoreDoneHMI, PT := t#5s); // TP
F_ALARM_SetDefinition(bAlarmTrigger := aAlarmPulse[nAlarmIndex].Q, nCategoryNo := 5, nMessageTypeNo := E_MessageType.GENERALSYSTEMWARNING, sTextMessage := 'MACHINE CONFIG SETTINGS BACKUP RESTORED', tAlarmTimout := t#0ms, bAlarmDefinitionEnable := TRUE, bInhibitReset := FALSE, bInternalReset := FALSE, aAlarmsSettings := gMessage.aAlarmsSettings, nAlarmIndex := nAlarmIndex, sMsgInfo := gMessage.stAlarmTable.aMsgHMI[nAlarmIndex], stMsgAux := gMessage.stAlarmTable.aMsgAux[nAlarmIndex]);

// NETWORK 31
// 'Conveyor Mode Active'
F_ALARM_SetDefinition(bAlarmTrigger := gDevice.stMachineConfig.bPassthrough AND NOT (gDevice.eMachineState = E_SYSTEM_MachineState.PASSTHROUGHACTIVE), nCategoryNo := 3, nMessageTypeNo := E_MessageType.GENERALSYSTEMWARNING, sTextMessage := 'TRACK AND TRACE SYSTEM DEACTIVATED', tAlarmTimout := t#0ms, bAlarmDefinitionEnable := TRUE, bInhibitReset := FALSE, bInternalReset := FALSE, aAlarmsSettings := gMessage.aAlarmsSettings, nAlarmIndex := nAlarmIndex, sMsgInfo := gMessage.stAlarmTable.aMsgHMI[nAlarmIndex], stMsgAux := gMessage.stAlarmTable.aMsgAux[nAlarmIndex]);

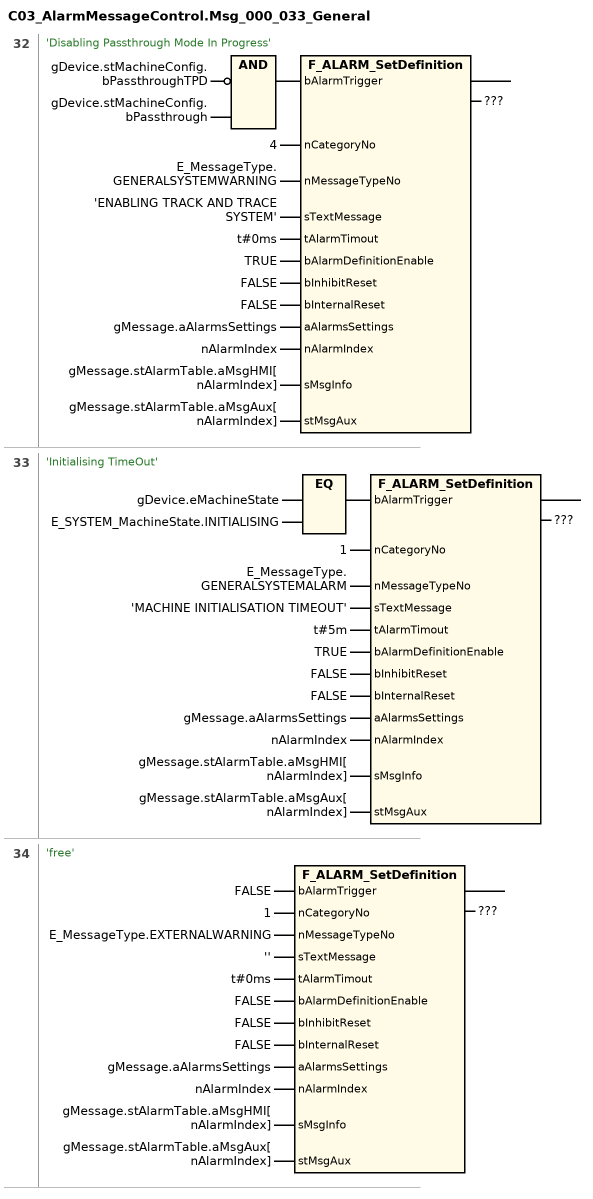
// NETWORK 32
// 'Disabling Passthrough Mode In Progress'
F_ALARM_SetDefinition(bAlarmTrigger := NOT gDevice.stMachineConfig.bPassthroughTPD AND gDevice.stMachineConfig.bPassthrough, nCategoryNo := 4, nMessageTypeNo := E_MessageType.GENERALSYSTEMWARNING, sTextMessage := 'ENABLING TRACK AND TRACE SYSTEM', tAlarmTimout := t#0ms, bAlarmDefinitionEnable := TRUE, bInhibitReset := FALSE, bInternalReset := FALSE, aAlarmsSettings := gMessage.aAlarmsSettings, nAlarmIndex := nAlarmIndex, sMsgInfo := gMessage.stAlarmTable.aMsgHMI[nAlarmIndex], stMsgAux := gMessage.stAlarmTable.aMsgAux[nAlarmIndex]);

// NETWORK 33
// 'Initialising TimeOut'
F_ALARM_SetDefinition(bAlarmTrigger := gDevice.eMachineState = E_SYSTEM_MachineState.INITIALISING, nCategoryNo := 1, nMessageTypeNo := E_MessageType.GENERALSYSTEMALARM, sTextMessage := 'MACHINE INITIALISATION TIMEOUT', tAlarmTimout := t#5m, bAlarmDefinitionEnable := TRUE, bInhibitReset := FALSE, bInternalReset := FALSE, aAlarmsSettings := gMessage.aAlarmsSettings, nAlarmIndex := nAlarmIndex, sMsgInfo := gMessage.stAlarmTable.aMsgHMI[nAlarmIndex], stMsgAux := gMessage.stAlarmTable.aMsgAux[nAlarmIndex]);

// NETWORK 34
// 'free'
F_ALARM_SetDefinition(bAlarmTrigger := FALSE, nCategoryNo := 1, nMessageTypeNo := E_MessageType.EXTERNALWARNING, sTextMessage := '', tAlarmTimout := t#0ms, bAlarmDefinitionEnable := FALSE, bInhibitReset := FALSE, bInternalReset := FALSE, aAlarmsSettings := gMessage.aAlarmsSettings, nAlarmIndex := nAlarmIndex, sMsgInfo := gMessage.stAlarmTable.aMsgHMI[nAlarmIndex], stMsgAux := gMessage.stAlarmTable.aMsgAux[nAlarmIndex]);
END_ACTION

ACTION Msg_034_074_Cameras:
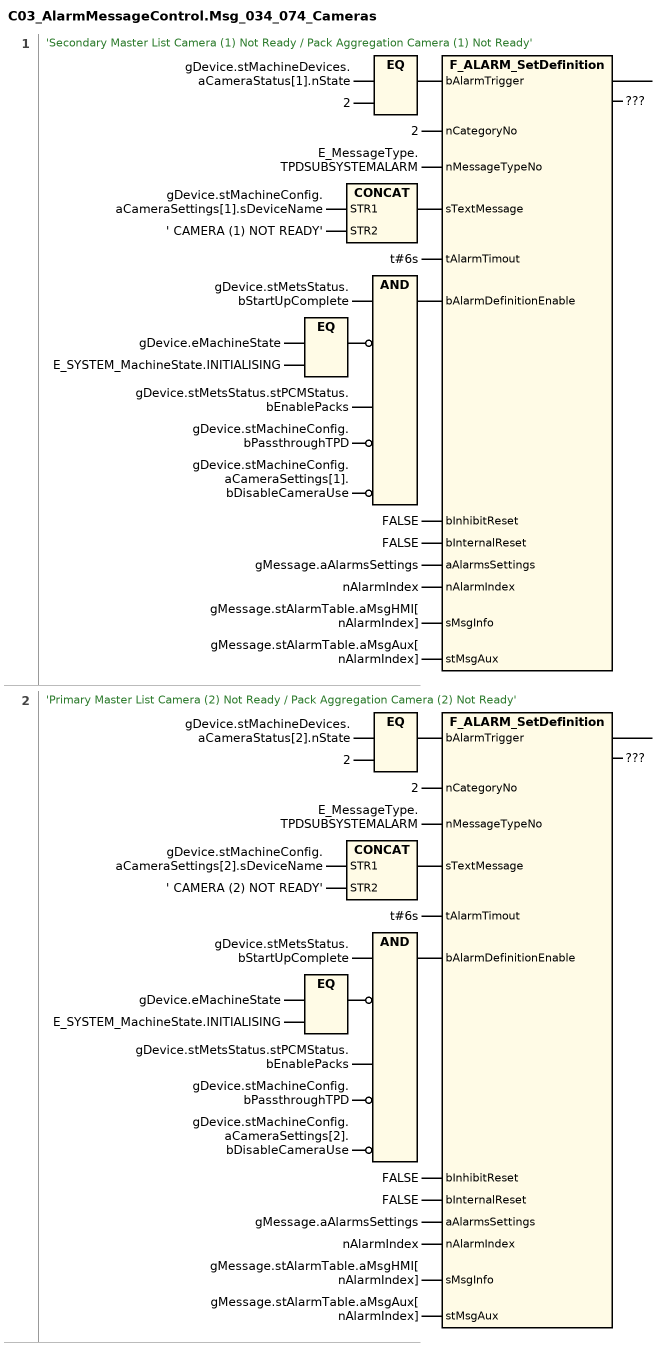
// NETWORK 1
// 'Secondary Master List Camera (1) Not Ready / Pack Aggregation Camera (1) Not Ready'
F_ALARM_SetDefinition(bAlarmTrigger := gDevice.stMachineDevices.aCameraStatus[1].nState = 2, nCategoryNo := 2, nMessageTypeNo := E_MessageType.TPDSUBSYSTEMALARM, sTextMessage := CONCAT(STR1 := gDevice.stMachineConfig.aCameraSettings[1].sDeviceName, STR2 := ' CAMERA (1) NOT READY'), tAlarmTimout := t#6s, bAlarmDefinitionEnable := gDevice.stMetsStatus.bStartUpComplete AND NOT (gDevice.eMachineState = E_SYSTEM_MachineState.INITIALISING) AND gDevice.stMetsStatus.stPCMStatus.bEnablePacks AND NOT gDevice.stMachineConfig.bPassthroughTPD AND NOT gDevice.stMachineConfig.aCameraSettings[1].bDisableCameraUse, bInhibitReset := FALSE, bInternalReset := FALSE, aAlarmsSettings := gMessage.aAlarmsSettings, nAlarmIndex := nAlarmIndex, sMsgInfo := gMessage.stAlarmTable.aMsgHMI[nAlarmIndex], stMsgAux := gMessage.stAlarmTable.aMsgAux[nAlarmIndex]);

// NETWORK 2
// 'Primary Master List Camera (2) Not Ready / Pack Aggregation Camera (2) Not Ready'
F_ALARM_SetDefinition(bAlarmTrigger := gDevice.stMachineDevices.aCameraStatus[2].nState = 2, nCategoryNo := 2, nMessageTypeNo := E_MessageType.TPDSUBSYSTEMALARM, sTextMessage := CONCAT(STR1 := gDevice.stMachineConfig.aCameraSettings[2].sDeviceName, STR2 := ' CAMERA (2) NOT READY'), tAlarmTimout := t#6s, bAlarmDefinitionEnable := gDevice.stMetsStatus.bStartUpComplete AND NOT (gDevice.eMachineState = E_SYSTEM_MachineState.INITIALISING) AND gDevice.stMetsStatus.stPCMStatus.bEnablePacks AND NOT gDevice.stMachineConfig.bPassthroughTPD AND NOT gDevice.stMachineConfig.aCameraSettings[2].bDisableCameraUse, bInhibitReset := FALSE, bInternalReset := FALSE, aAlarmsSettings := gMessage.aAlarmsSettings, nAlarmIndex := nAlarmIndex, sMsgInfo := gMessage.stAlarmTable.aMsgHMI[nAlarmIndex], stMsgAux := gMessage.stAlarmTable.aMsgAux[nAlarmIndex]);

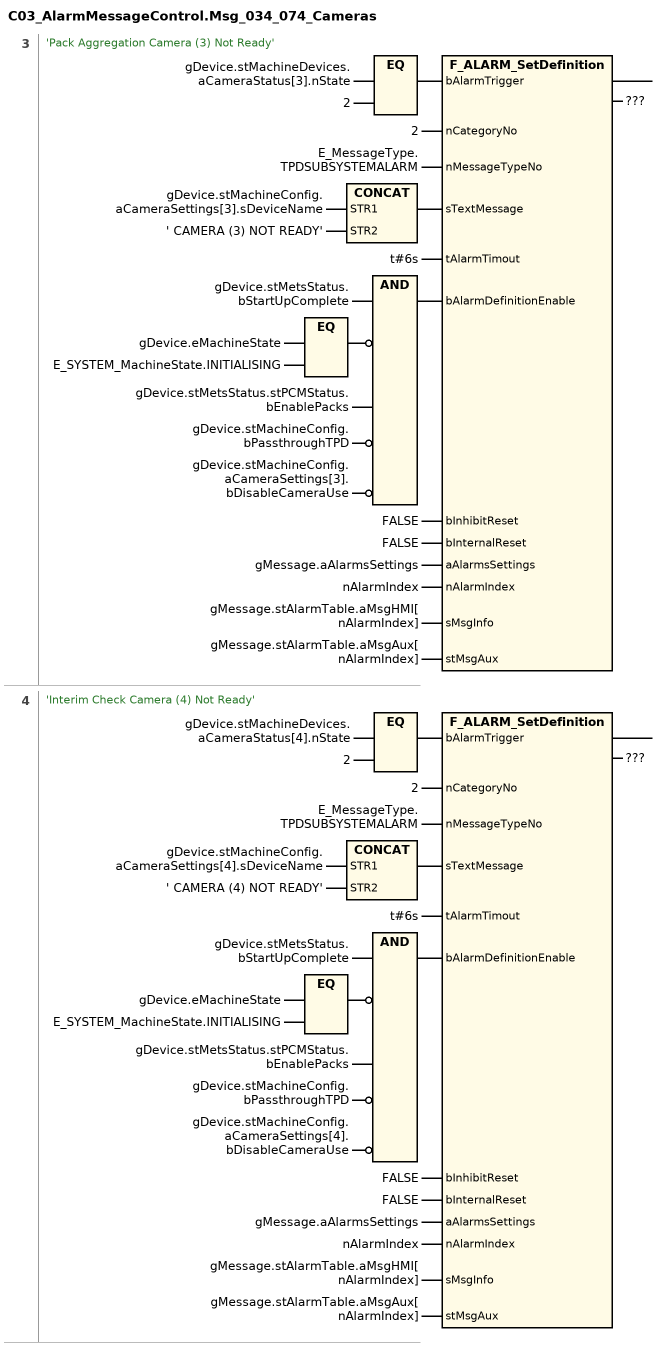
// NETWORK 3
// 'Pack Aggregation Camera (3) Not Ready'
F_ALARM_SetDefinition(bAlarmTrigger := gDevice.stMachineDevices.aCameraStatus[3].nState = 2, nCategoryNo := 2, nMessageTypeNo := E_MessageType.TPDSUBSYSTEMALARM, sTextMessage := CONCAT(STR1 := gDevice.stMachineConfig.aCameraSettings[3].sDeviceName, STR2 := ' CAMERA (3) NOT READY'), tAlarmTimout := t#6s, bAlarmDefinitionEnable := gDevice.stMetsStatus.bStartUpComplete AND NOT (gDevice.eMachineState = E_SYSTEM_MachineState.INITIALISING) AND gDevice.stMetsStatus.stPCMStatus.bEnablePacks AND NOT gDevice.stMachineConfig.bPassthroughTPD AND NOT gDevice.stMachineConfig.aCameraSettings[3].bDisableCameraUse, bInhibitReset := FALSE, bInternalReset := FALSE, aAlarmsSettings := gMessage.aAlarmsSettings, nAlarmIndex := nAlarmIndex, sMsgInfo := gMessage.stAlarmTable.aMsgHMI[nAlarmIndex], stMsgAux := gMessage.stAlarmTable.aMsgAux[nAlarmIndex]);

// NETWORK 4
// 'Interim Check Camera (4) Not Ready'
F_ALARM_SetDefinition(bAlarmTrigger := gDevice.stMachineDevices.aCameraStatus[4].nState = 2, nCategoryNo := 2, nMessageTypeNo := E_MessageType.TPDSUBSYSTEMALARM, sTextMessage := CONCAT(STR1 := gDevice.stMachineConfig.aCameraSettings[4].sDeviceName, STR2 := ' CAMERA (4) NOT READY'), tAlarmTimout := t#6s, bAlarmDefinitionEnable := gDevice.stMetsStatus.bStartUpComplete AND NOT (gDevice.eMachineState = E_SYSTEM_MachineState.INITIALISING) AND gDevice.stMetsStatus.stPCMStatus.bEnablePacks AND NOT gDevice.stMachineConfig.bPassthroughTPD AND NOT gDevice.stMachineConfig.aCameraSettings[4].bDisableCameraUse, bInhibitReset := FALSE, bInternalReset := FALSE, aAlarmsSettings := gMessage.aAlarmsSettings, nAlarmIndex := nAlarmIndex, sMsgInfo := gMessage.stAlarmTable.aMsgHMI[nAlarmIndex], stMsgAux := gMessage.stAlarmTable.aMsgAux[nAlarmIndex]);

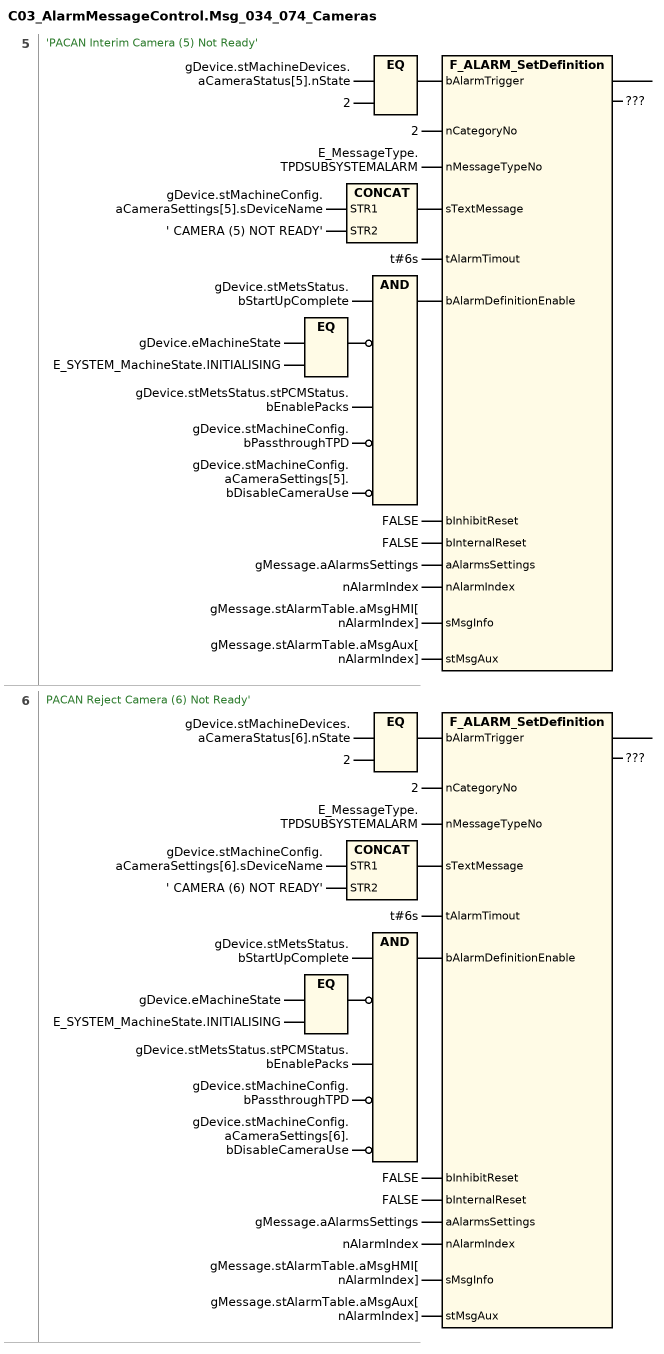
// NETWORK 5
// 'PACAN Interim Camera (5) Not Ready'
F_ALARM_SetDefinition(bAlarmTrigger := gDevice.stMachineDevices.aCameraStatus[5].nState = 2, nCategoryNo := 2, nMessageTypeNo := E_MessageType.TPDSUBSYSTEMALARM, sTextMessage := CONCAT(STR1 := gDevice.stMachineConfig.aCameraSettings[5].sDeviceName, STR2 := ' CAMERA (5) NOT READY'), tAlarmTimout := t#6s, bAlarmDefinitionEnable := gDevice.stMetsStatus.bStartUpComplete AND NOT (gDevice.eMachineState = E_SYSTEM_MachineState.INITIALISING) AND gDevice.stMetsStatus.stPCMStatus.bEnablePacks AND NOT gDevice.stMachineConfig.bPassthroughTPD AND NOT gDevice.stMachineConfig.aCameraSettings[5].bDisableCameraUse, bInhibitReset := FALSE, bInternalReset := FALSE, aAlarmsSettings := gMessage.aAlarmsSettings, nAlarmIndex := nAlarmIndex, sMsgInfo := gMessage.stAlarmTable.aMsgHMI[nAlarmIndex], stMsgAux := gMessage.stAlarmTable.aMsgAux[nAlarmIndex]);

// NETWORK 6
// PACAN Reject Camera (6) Not Ready'
F_ALARM_SetDefinition(bAlarmTrigger := gDevice.stMachineDevices.aCameraStatus[6].nState = 2, nCategoryNo := 2, nMessageTypeNo := E_MessageType.TPDSUBSYSTEMALARM, sTextMessage := CONCAT(STR1 := gDevice.stMachineConfig.aCameraSettings[6].sDeviceName, STR2 := ' CAMERA (6) NOT READY'), tAlarmTimout := t#6s, bAlarmDefinitionEnable := gDevice.stMetsStatus.bStartUpComplete AND NOT (gDevice.eMachineState = E_SYSTEM_MachineState.INITIALISING) AND gDevice.stMetsStatus.stPCMStatus.bEnablePacks AND NOT gDevice.stMachineConfig.bPassthroughTPD AND NOT gDevice.stMachineConfig.aCameraSettings[6].bDisableCameraUse, bInhibitReset := FALSE, bInternalReset := FALSE, aAlarmsSettings := gMessage.aAlarmsSettings, nAlarmIndex := nAlarmIndex, sMsgInfo := gMessage.stAlarmTable.aMsgHMI[nAlarmIndex], stMsgAux := gMessage.stAlarmTable.aMsgAux[nAlarmIndex]);

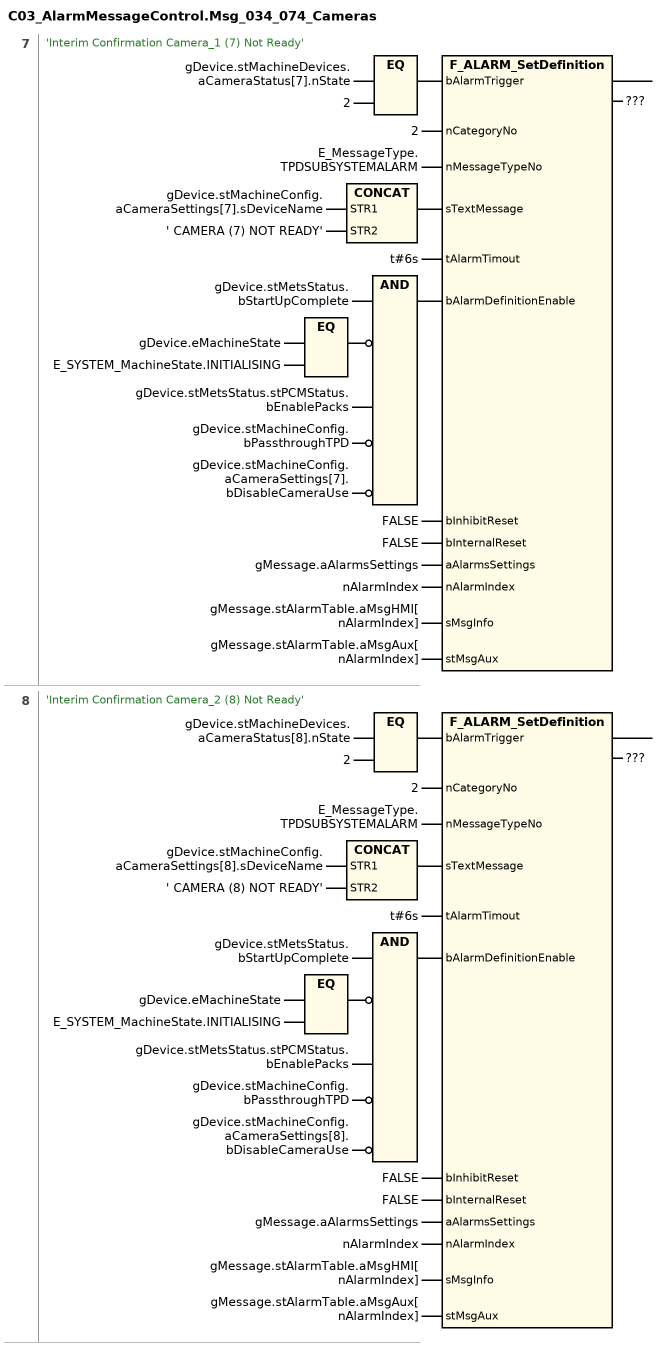
// NETWORK 7
// 'Interim Confirmation Camera_1 (7) Not Ready'
F_ALARM_SetDefinition(bAlarmTrigger := gDevice.stMachineDevices.aCameraStatus[7].nState = 2, nCategoryNo := 2, nMessageTypeNo := E_MessageType.TPDSUBSYSTEMALARM, sTextMessage := CONCAT(STR1 := gDevice.stMachineConfig.aCameraSettings[7].sDeviceName, STR2 := ' CAMERA (7) NOT READY'), tAlarmTimout := t#6s, bAlarmDefinitionEnable := gDevice.stMetsStatus.bStartUpComplete AND NOT (gDevice.eMachineState = E_SYSTEM_MachineState.INITIALISING) AND gDevice.stMetsStatus.stPCMStatus.bEnablePacks AND NOT gDevice.stMachineConfig.bPassthroughTPD AND NOT gDevice.stMachineConfig.aCameraSettings[7].bDisableCameraUse, bInhibitReset := FALSE, bInternalReset := FALSE, aAlarmsSettings := gMessage.aAlarmsSettings, nAlarmIndex := nAlarmIndex, sMsgInfo := gMessage.stAlarmTable.aMsgHMI[nAlarmIndex], stMsgAux := gMessage.stAlarmTable.aMsgAux[nAlarmIndex]);

// NETWORK 8
// 'Interim Confirmation Camera_2 (8) Not Ready'
F_ALARM_SetDefinition(bAlarmTrigger := gDevice.stMachineDevices.aCameraStatus[8].nState = 2, nCategoryNo := 2, nMessageTypeNo := E_MessageType.TPDSUBSYSTEMALARM, sTextMessage := CONCAT(STR1 := gDevice.stMachineConfig.aCameraSettings[8].sDeviceName, STR2 := ' CAMERA (8) NOT READY'), tAlarmTimout := t#6s, bAlarmDefinitionEnable := gDevice.stMetsStatus.bStartUpComplete AND NOT (gDevice.eMachineState = E_SYSTEM_MachineState.INITIALISING) AND gDevice.stMetsStatus.stPCMStatus.bEnablePacks AND NOT gDevice.stMachineConfig.bPassthroughTPD AND NOT gDevice.stMachineConfig.aCameraSettings[8].bDisableCameraUse, bInhibitReset := FALSE, bInternalReset := FALSE, aAlarmsSettings := gMessage.aAlarmsSettings, nAlarmIndex := nAlarmIndex, sMsgInfo := gMessage.stAlarmTable.aMsgHMI[nAlarmIndex], stMsgAux := gMessage.stAlarmTable.aMsgAux[nAlarmIndex]);

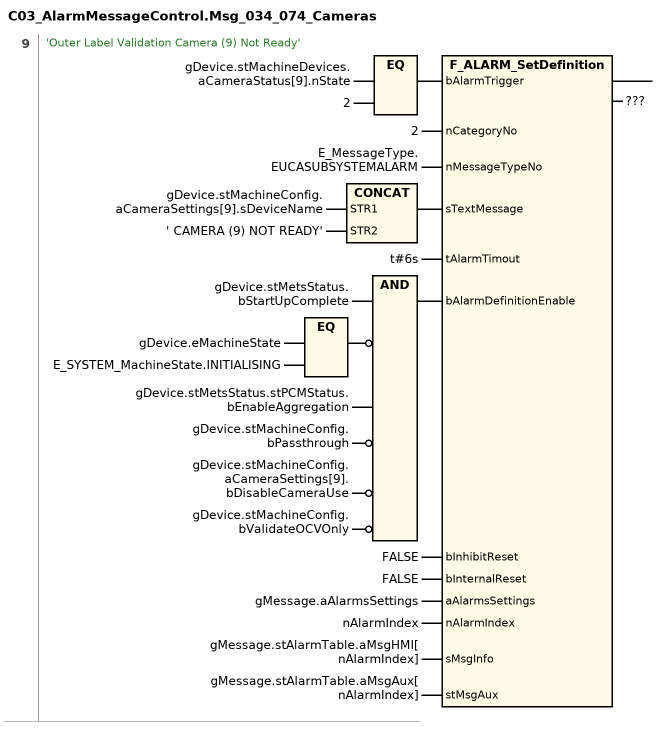
// NETWORK 9
// 'Outer Label Validation Camera (9) Not Ready'
F_ALARM_SetDefinition(bAlarmTrigger := gDevice.stMachineDevices.aCameraStatus[9].nState = 2, nCategoryNo := 2, nMessageTypeNo := E_MessageType.EUCASUBSYSTEMALARM, sTextMessage := CONCAT(STR1 := gDevice.stMachineConfig.aCameraSettings[9].sDeviceName, STR2 := ' CAMERA (9) NOT READY'), tAlarmTimout := t#6s, bAlarmDefinitionEnable := gDevice.stMetsStatus.bStartUpComplete AND NOT (gDevice.eMachineState = E_SYSTEM_MachineState.INITIALISING) AND gDevice.stMetsStatus.stPCMStatus.bEnableAggregation AND NOT gDevice.stMachineConfig.bPassthrough AND NOT gDevice.stMachineConfig.aCameraSettings[9].bDisableCameraUse AND NOT gDevice.stMachineConfig.bValidateOCVOnly, bInhibitReset := FALSE, bInternalReset := FALSE, aAlarmsSettings := gMessage.aAlarmsSettings, nAlarmIndex := nAlarmIndex, sMsgInfo := gMessage.stAlarmTable.aMsgHMI[nAlarmIndex], stMsgAux := gMessage.stAlarmTable.aMsgAux[nAlarmIndex]);

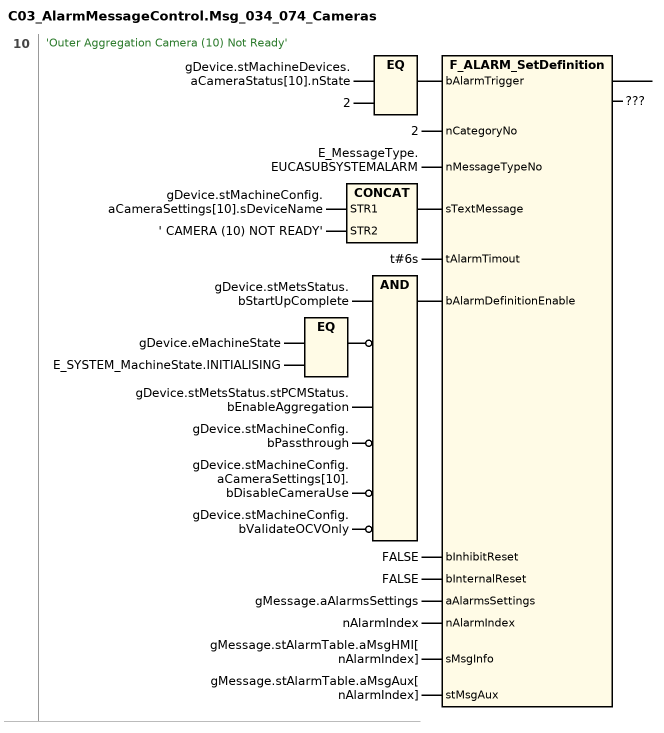
// NETWORK 10
// 'Outer Aggregation Camera (10) Not Ready'
F_ALARM_SetDefinition(bAlarmTrigger := gDevice.stMachineDevices.aCameraStatus[10].nState = 2, nCategoryNo := 2, nMessageTypeNo := E_MessageType.EUCASUBSYSTEMALARM, sTextMessage := CONCAT(STR1 := gDevice.stMachineConfig.aCameraSettings[10].sDeviceName, STR2 := ' CAMERA (10) NOT READY'), tAlarmTimout := t#6s, bAlarmDefinitionEnable := gDevice.stMetsStatus.bStartUpComplete AND NOT (gDevice.eMachineState = E_SYSTEM_MachineState.INITIALISING) AND gDevice.stMetsStatus.stPCMStatus.bEnableAggregation AND NOT gDevice.stMachineConfig.bPassthrough AND NOT gDevice.stMachineConfig.aCameraSettings[10].bDisableCameraUse AND NOT gDevice.stMachineConfig.bValidateOCVOnly, bInhibitReset := FALSE, bInternalReset := FALSE, aAlarmsSettings := gMessage.aAlarmsSettings, nAlarmIndex := nAlarmIndex, sMsgInfo := gMessage.stAlarmTable.aMsgHMI[nAlarmIndex], stMsgAux := gMessage.stAlarmTable.aMsgAux[nAlarmIndex]);

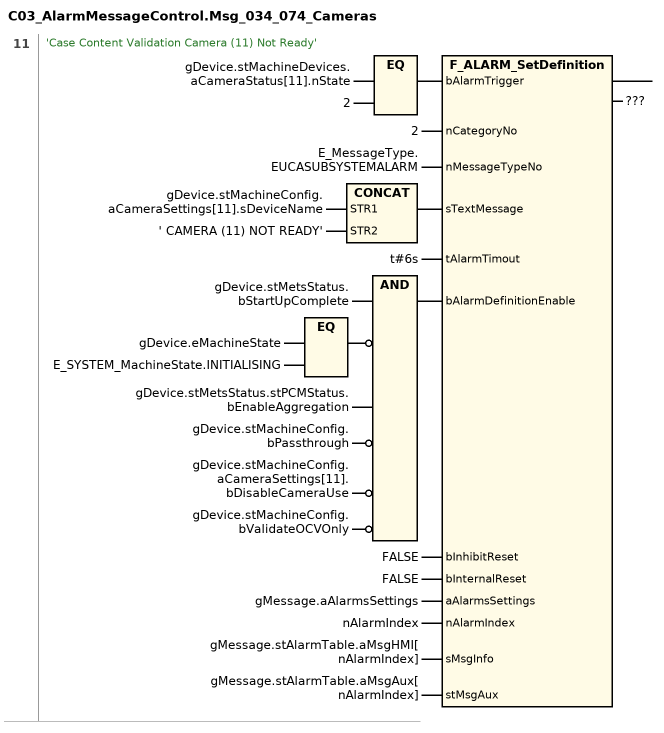
// NETWORK 11
// 'Case Content Validation Camera (11) Not Ready'
F_ALARM_SetDefinition(bAlarmTrigger := gDevice.stMachineDevices.aCameraStatus[11].nState = 2, nCategoryNo := 2, nMessageTypeNo := E_MessageType.EUCASUBSYSTEMALARM, sTextMessage := CONCAT(STR1 := gDevice.stMachineConfig.aCameraSettings[11].sDeviceName, STR2 := ' CAMERA (11) NOT READY'), tAlarmTimout := t#6s, bAlarmDefinitionEnable := gDevice.stMetsStatus.bStartUpComplete AND NOT (gDevice.eMachineState = E_SYSTEM_MachineState.INITIALISING) AND gDevice.stMetsStatus.stPCMStatus.bEnableAggregation AND NOT gDevice.stMachineConfig.bPassthrough AND NOT gDevice.stMachineConfig.aCameraSettings[11].bDisableCameraUse AND NOT gDevice.stMachineConfig.bValidateOCVOnly, bInhibitReset := FALSE, bInternalReset := FALSE, aAlarmsSettings := gMessage.aAlarmsSettings, nAlarmIndex := nAlarmIndex, sMsgInfo := gMessage.stAlarmTable.aMsgHMI[nAlarmIndex], stMsgAux := gMessage.stAlarmTable.aMsgAux[nAlarmIndex]);

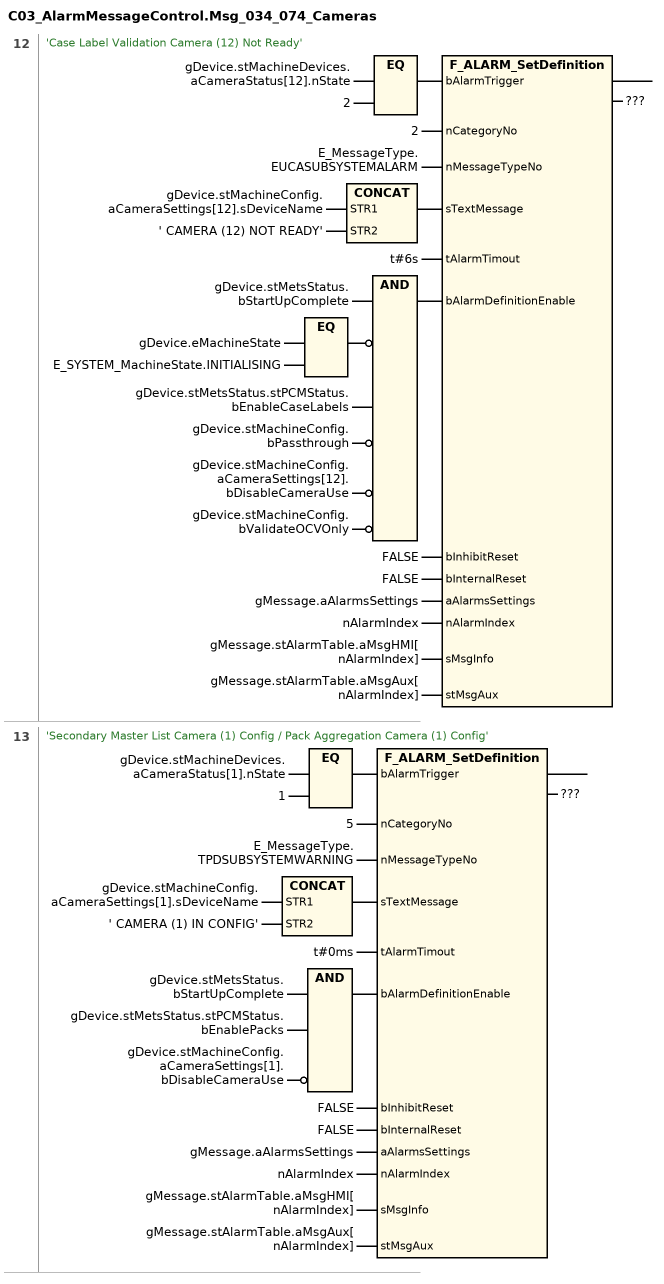
// NETWORK 12
// 'Case Label Validation Camera (12) Not Ready'
F_ALARM_SetDefinition(bAlarmTrigger := gDevice.stMachineDevices.aCameraStatus[12].nState = 2, nCategoryNo := 2, nMessageTypeNo := E_MessageType.EUCASUBSYSTEMALARM, sTextMessage := CONCAT(STR1 := gDevice.stMachineConfig.aCameraSettings[12].sDeviceName, STR2 := ' CAMERA (12) NOT READY'), tAlarmTimout := t#6s, bAlarmDefinitionEnable := gDevice.stMetsStatus.bStartUpComplete AND NOT (gDevice.eMachineState = E_SYSTEM_MachineState.INITIALISING) AND gDevice.stMetsStatus.stPCMStatus.bEnableCaseLabels AND NOT gDevice.stMachineConfig.bPassthrough AND NOT gDevice.stMachineConfig.aCameraSettings[12].bDisableCameraUse AND NOT gDevice.stMachineConfig.bValidateOCVOnly, bInhibitReset := FALSE, bInternalReset := FALSE, aAlarmsSettings := gMessage.aAlarmsSettings, nAlarmIndex := nAlarmIndex, sMsgInfo := gMessage.stAlarmTable.aMsgHMI[nAlarmIndex], stMsgAux := gMessage.stAlarmTable.aMsgAux[nAlarmIndex]);

// NETWORK 13
// 'Secondary Master List Camera (1) Config / Pack Aggregation Camera (1) Config'
F_ALARM_SetDefinition(bAlarmTrigger := gDevice.stMachineDevices.aCameraStatus[1].nState = 1, nCategoryNo := 5, nMessageTypeNo := E_MessageType.TPDSUBSYSTEMWARNING, sTextMessage := CONCAT(STR1 := gDevice.stMachineConfig.aCameraSettings[1].sDeviceName, STR2 := ' CAMERA (1) IN CONFIG'), tAlarmTimout := t#0ms, bAlarmDefinitionEnable := gDevice.stMetsStatus.bStartUpComplete AND gDevice.stMetsStatus.stPCMStatus.bEnablePacks AND NOT gDevice.stMachineConfig.aCameraSettings[1].bDisableCameraUse, bInhibitReset := FALSE, bInternalReset := FALSE, aAlarmsSettings := gMessage.aAlarmsSettings, nAlarmIndex := nAlarmIndex, sMsgInfo := gMessage.stAlarmTable.aMsgHMI[nAlarmIndex], stMsgAux := gMessage.stAlarmTable.aMsgAux[nAlarmIndex]);

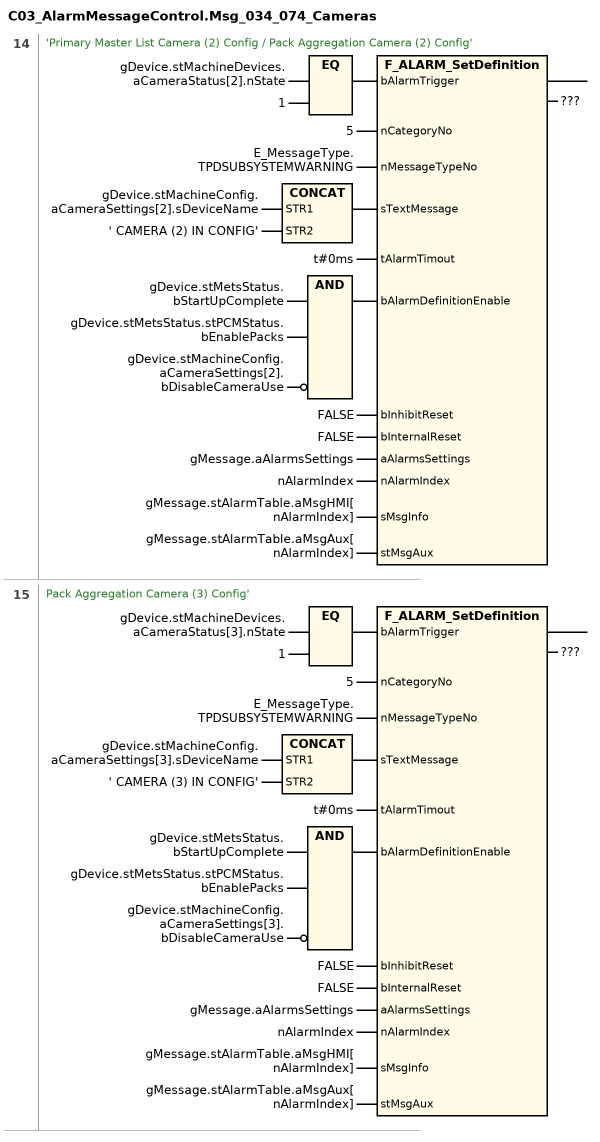
// NETWORK 14
// 'Primary Master List Camera (2) Config / Pack Aggregation Camera (2) Config'
F_ALARM_SetDefinition(bAlarmTrigger := gDevice.stMachineDevices.aCameraStatus[2].nState = 1, nCategoryNo := 5, nMessageTypeNo := E_MessageType.TPDSUBSYSTEMWARNING, sTextMessage := CONCAT(STR1 := gDevice.stMachineConfig.aCameraSettings[2].sDeviceName, STR2 := ' CAMERA (2) IN CONFIG'), tAlarmTimout := t#0ms, bAlarmDefinitionEnable := gDevice.stMetsStatus.bStartUpComplete AND gDevice.stMetsStatus.stPCMStatus.bEnablePacks AND NOT gDevice.stMachineConfig.aCameraSettings[2].bDisableCameraUse, bInhibitReset := FALSE, bInternalReset := FALSE, aAlarmsSettings := gMessage.aAlarmsSettings, nAlarmIndex := nAlarmIndex, sMsgInfo := gMessage.stAlarmTable.aMsgHMI[nAlarmIndex], stMsgAux := gMessage.stAlarmTable.aMsgAux[nAlarmIndex]);

// NETWORK 15
// Pack Aggregation Camera (3) Config'
F_ALARM_SetDefinition(bAlarmTrigger := gDevice.stMachineDevices.aCameraStatus[3].nState = 1, nCategoryNo := 5, nMessageTypeNo := E_MessageType.TPDSUBSYSTEMWARNING, sTextMessage := CONCAT(STR1 := gDevice.stMachineConfig.aCameraSettings[3].sDeviceName, STR2 := ' CAMERA (3) IN CONFIG'), tAlarmTimout := t#0ms, bAlarmDefinitionEnable := gDevice.stMetsStatus.bStartUpComplete AND gDevice.stMetsStatus.stPCMStatus.bEnablePacks AND NOT gDevice.stMachineConfig.aCameraSettings[3].bDisableCameraUse, bInhibitReset := FALSE, bInternalReset := FALSE, aAlarmsSettings := gMessage.aAlarmsSettings, nAlarmIndex := nAlarmIndex, sMsgInfo := gMessage.stAlarmTable.aMsgHMI[nAlarmIndex], stMsgAux := gMessage.stAlarmTable.aMsgAux[nAlarmIndex]);

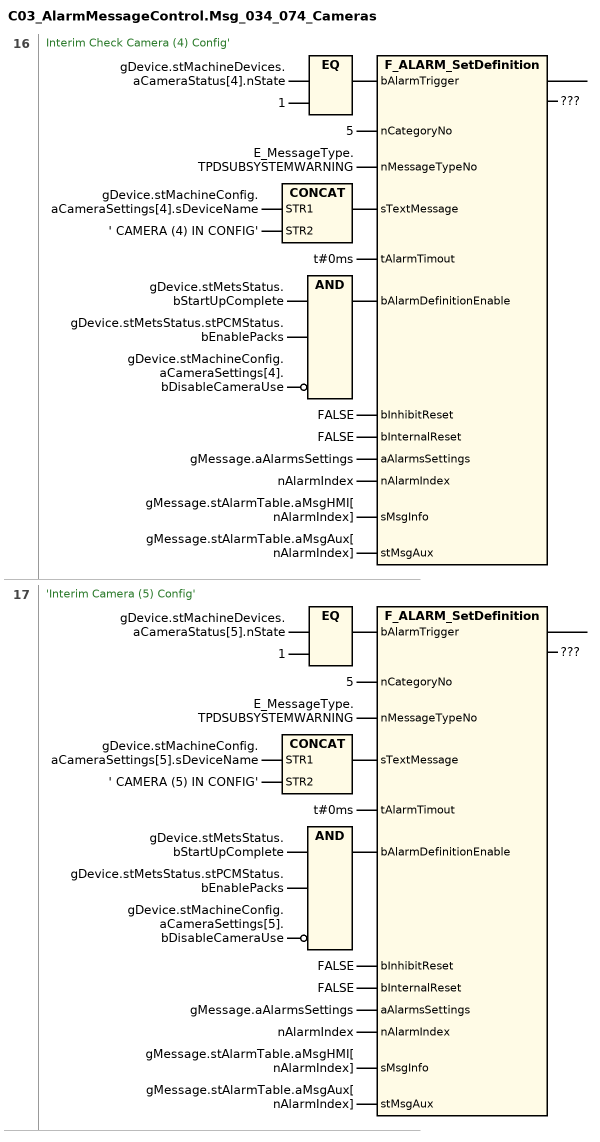
// NETWORK 16
// Interim Check Camera (4) Config'
F_ALARM_SetDefinition(bAlarmTrigger := gDevice.stMachineDevices.aCameraStatus[4].nState = 1, nCategoryNo := 5, nMessageTypeNo := E_MessageType.TPDSUBSYSTEMWARNING, sTextMessage := CONCAT(STR1 := gDevice.stMachineConfig.aCameraSettings[4].sDeviceName, STR2 := ' CAMERA (4) IN CONFIG'), tAlarmTimout := t#0ms, bAlarmDefinitionEnable := gDevice.stMetsStatus.bStartUpComplete AND gDevice.stMetsStatus.stPCMStatus.bEnablePacks AND NOT gDevice.stMachineConfig.aCameraSettings[4].bDisableCameraUse, bInhibitReset := FALSE, bInternalReset := FALSE, aAlarmsSettings := gMessage.aAlarmsSettings, nAlarmIndex := nAlarmIndex, sMsgInfo := gMessage.stAlarmTable.aMsgHMI[nAlarmIndex], stMsgAux := gMessage.stAlarmTable.aMsgAux[nAlarmIndex]);

// NETWORK 17
// 'Interim Camera (5) Config'
F_ALARM_SetDefinition(bAlarmTrigger := gDevice.stMachineDevices.aCameraStatus[5].nState = 1, nCategoryNo := 5, nMessageTypeNo := E_MessageType.TPDSUBSYSTEMWARNING, sTextMessage := CONCAT(STR1 := gDevice.stMachineConfig.aCameraSettings[5].sDeviceName, STR2 := ' CAMERA (5) IN CONFIG'), tAlarmTimout := t#0ms, bAlarmDefinitionEnable := gDevice.stMetsStatus.bStartUpComplete AND gDevice.stMetsStatus.stPCMStatus.bEnablePacks AND NOT gDevice.stMachineConfig.aCameraSettings[5].bDisableCameraUse, bInhibitReset := FALSE, bInternalReset := FALSE, aAlarmsSettings := gMessage.aAlarmsSettings, nAlarmIndex := nAlarmIndex, sMsgInfo := gMessage.stAlarmTable.aMsgHMI[nAlarmIndex], stMsgAux := gMessage.stAlarmTable.aMsgAux[nAlarmIndex]);

